// TwinCAT 3 PLC project TPR
// libraries:
//   Tc2_Standard, * (Beckhoff Automation GmbH)
//   Tc2_System, * (Beckhoff Automation GmbH)
//   Tc2_Utilities, * (Beckhoff Automation GmbH)
//   Tc3_Database, * (Beckhoff Automation GmbH)
//   Tc3_EventLogger, * (Beckhoff Automation GmbH)
//   Tc3_IotBase, * (Beckhoff Automation GmbH)
//   Tc3_Module, * (Beckhoff Automation GmbH)
// project tree:
//   Data types/ PrgData.TcDUT, frameData.TcDUT, ST_DataFromVision.TcDUT, ST_DataToVision.TcDUT, ST_ToolControl.TcDUT, ST_ToolData.TcDUT, ST_AdsTest.TcDUT
//   Global Variables/ CartControls.TcGVL, ErrorVar.TcGVL, Global_Variables.TcGVL
//   / PLC.TcTTO
//   POUs/ BackToZero.TcPOU, DB_Conn.TcPOU, ErrorHandle.TcPOU, GetCoordinates.TcPOU, LogProgram.TcPOU, MAIN.TcPOU, OnOffRobotCut.TcPOU, PcCom.TcPOU, P_Mqtt.TcPOU, RobotService.TcPOU, SendCoordinates.TcPOU, Tools.TcPOU
//   POUs/CONTROLs/ BlockTest.TcPOU, CalibCam1.TcPOU, CalibCam2.TcPOU, Control.TcPOU, ControlAuto.TcPOU, ControlGrabAuto.TcPOU, ControlMoveToCalibPos.TcPOU
//   POUs/EasySql/F_FB/ FB_EasySql.TcPOU, F_Replace.TcPOU
//   POUs/FUNCTIONs/ CamControl_1.TcPOU, CamControl_2.TcPOU, PlaceCoordinates.TcPOU, RobotControl_1.TcPOU, ValveControl_1.TcPOU
//   POUs/SEQUENCEs/ DeleafPlace.TcPOU, FindJoint.TcPOU, GetStem.TcPOU, GrabJoint.TcPOU, GrabStem.TcPOU, MoveOnStem.TcPOU
//   POUs/SQL/00_TestData/ P_SqlGeneratTestData.TcPOU
//   POUs/SQL/01_Insert/ P_SqlInsert.TcPOU, P_SqlInsertLog.TcPOU, P_SqlInsertRowConstructor.TcPOU, P_SqlInsertUnionAll.TcPOU, P_SqlInsertAlarmLog.TcPOU
//   POUs/SQL/02_Delete/ P_SqlDelete.TcPOU
//   POUs/SQL/03_Select/ P_SqlSelect.TcPOU, P_SqlSelectAlarmLog.TcPOU, P_SqlSelectCurrent.TcPOU, P_SqlSelectAlarm.TcPOU, P_SqlSelectTop.TcPOU, P_SqlSelectRecipe.TcPOU, P_SqlSelectFrame.TcPOU, ST_SelectAlarmStruct.TcDUT, ST_SelectAlarmLogStruct.TcDUT, ST_SelectFrameStruct.TcDUT, ST_SelectCurrentStruct.TcDUT, ST_SelectStruct.TcDUT, ST_SelectRecipeStruct.TcDUT
//   POUs/SQL/04_Update/ P_SqlUpdate.TcPOU, P_SqlUpdateAlarmLog.TcPOU
//   POUs/SQL/05_Count/ P_SqlCount.TcPOU
//   POUs/SQL/06_Sum/ P_SqlSum.TcPOU
// real-time tasks:
//   TASK PLC: cycle T#10ms, priority 1, ADS port 350
// I/O:
//   DEVICE Device 1 (Beckhoff CCAT)
//   DEVICE Device 2 (EtherCAT), AmsNetId 192.168.56.1.3.1
//     Term 1 (EK1200) [EK1200-5000 EtherCAT Power supply (2A E-Bus)]
//       Term 2 (EL1859) [EL1859 8Ch. Dig. Input 24V, 3ms, 8Ch. Dig. Output 24V, 0.5A]
//       Term 3 (EL2809) [EL2809 16Ch. Dig. Output 24V, 0.5A]
//       Term 4 (EL5151) [EL5151 1Ch. Inc. Encoder]
//       Term 5 (EL6751) [EL6751 CANopen Master]
//       Term 6 (EL9011) [EL9011 End Terminal]
//   DEVICE Device 3 (EL6751), AmsNetId 192.168.56.1.4.1
//     Box 7 (CX2xxx CANopen Slave)
// variable links:
//   TPR/TPR Instance <-> Device 2 (EtherCAT)/Term 1 (EK1200)/Term 2 (EL1859)
//     PLC Inputs/Global_Variables.bGripSensorStop <-> Channel 2/Input
//     PLC Inputs/OnOffRobotCut.bStartBotton <-> Channel 1/Input
//     PLC Outputs/Tools.qValve1 <-> Channel 9/Output
//     PLC Outputs/Tools.qValve2 <-> Channel 10/Output
//     PLC Outputs/Tools.qValve3 <-> Channel 11/Output
//     PLC Outputs/Tools.qValve4 <-> Channel 13/Output
//     PLC Outputs/Tools.qValve5 <-> Channel 12/Output
//   TPR/TPR Instance <-> Device 2 (EtherCAT)/Term 1 (EK1200)/Term 3 (EL2809)
//     PLC Outputs/CartControls.CartBackward <-> Channel 8/Output
//     PLC Outputs/CartControls.CartDown <-> Channel 6/Output
//     PLC Outputs/CartControls.CartForward <-> Channel 7/Output
//     PLC Outputs/CartControls.CartUp <-> Channel 5/Output
//     PLC Outputs/CartControls.WheelsChange <-> Channel 10/Output
//     PLC Outputs/Tools.qMotorDirection <-> Channel 2/Output
//     PLC Outputs/Tools.qMotorRun <-> Channel 1/Output
//   TPR/TPR Instance <-> Device 2 (EtherCAT)/Term 1 (EK1200)/Term 4 (EL5151)
//     PLC Inputs/Global_Variables.uiSignalInEncoderCount <-> ENC Inputs/Counter value
//     PLC Outputs/Global_Variables.bSetCounter <-> ENC Outputs/Control/Set counter
//     PLC Outputs/Global_Variables.uiSetCounterValue <-> ENC Outputs/Set counter value
//   TPR/TPR Instance <-> Device 3 (EL6751)/Box 7 (CX2xxx CANopen Slave)
//     PLC Inputs/ErrorVar.ErrorNum <-> TxPDO 4/Inputs/Byte_Input_30
//     PLC Inputs/ErrorVar.ErrorNum @bit 8 <-> TxPDO 4/Inputs/Byte_Input_31
//     PLC Inputs/ErrorVar.ErrorNum @bit 16 <-> TxPDO 4/Inputs/Byte_Input_32
//     PLC Inputs/ErrorVar.WhichRobot <-> TxPDO 4/Inputs/Byte_Input_29
//     PLC Inputs/Global_Variables.uiSignalIn2 <-> TxPDO 1/Inputs/Byte_Input_2
//     PLC Inputs/Global_Variables.uiSignalIn4 <-> TxPDO 1/Inputs/Byte_Input_4
//     PLC Inputs/Global_Variables.uiSignalInA <-> TxPDO 2/Inputs/Byte_Input_13
//     PLC Inputs/Global_Variables.uiSignalInA @bit 8 <-> TxPDO 2/Inputs/Byte_Input_14
//     PLC Inputs/Global_Variables.uiSignalInAck <-> TxPDO 1/Inputs/Byte_Input_5
//     PLC Inputs/Global_Variables.uiSignalInE <-> TxPDO 2/Inputs/Byte_Input_15
//     PLC Inputs/Global_Variables.uiSignalInE @bit 8 <-> TxPDO 2/Inputs/Byte_Input_16
//     PLC Inputs/Global_Variables.uiSignalInOrientation <-> TxPDO 3/Inputs/Byte_Input_19
//     PLC Inputs/Global_Variables.uiSignalInR <-> TxPDO 3/Inputs/Byte_Input_17
//     PLC Inputs/Global_Variables.uiSignalInR @bit 8 <-> TxPDO 3/Inputs/Byte_Input_18
//     PLC Inputs/Global_Variables.uiSignalInRobotFail <-> TxPDO 4/Inputs/Byte_Input_27
//     PLC Inputs/Global_Variables.uiSignalInShared <-> TxPDO 2/Inputs/Byte_Input_12
//     PLC Inputs/Global_Variables.uiSignalInToolAck <-> TxPDO 3/Inputs/Byte_Input_20
//     PLC Inputs/Global_Variables.uiSignalInX <-> TxPDO 3/Inputs/Byte_Input_21
//     PLC Inputs/Global_Variables.uiSignalInX @bit 8 <-> TxPDO 3/Inputs/Byte_Input_22
//     PLC Inputs/Global_Variables.uiSignalInY <-> TxPDO 3/Inputs/Byte_Input_23
//     PLC Inputs/Global_Variables.uiSignalInY @bit 8 <-> TxPDO 3/Inputs/Byte_Input_24
//     PLC Inputs/Global_Variables.uiSignalInZ <-> TxPDO 4/Inputs/Byte_Input_25
//     PLC Inputs/Global_Variables.uiSignalInZ @bit 8 <-> TxPDO 4/Inputs/Byte_Input_26
//     PLC Inputs/OnOffRobotCut.uiSignalIn1 <-> TxPDO 1/Inputs/Byte_Input_1
//     PLC Inputs/OnOffRobotCut.uiSignalIn3 <-> TxPDO 1/Inputs/Byte_Input_3
//     PLC Outputs/ErrorVar.CancelAlarm <-> RxPDO 4/Outputs/Byte_Output_32
//     PLC Outputs/ErrorVar.gSeverity <-> RxPDO 4/Outputs/Byte_Output_31
//     PLC Outputs/Global_Variables.gJointFound <-> RxPDO 3/Outputs/Byte_Output_18
//     PLC Outputs/Global_Variables.gTomatoHeading <-> RxPDO 4/Outputs/Byte_Output_29
//     PLC Outputs/Global_Variables.iImageZone <-> RxPDO 2/Outputs/Byte_Output_16
//     PLC Outputs/Global_Variables.uiCalibImgCount <-> RxPDO 2/Outputs/Byte_Output_14
//     PLC Outputs/Global_Variables.uiSignalOut1 <-> RxPDO 1/Outputs/Byte_Output_1
//     PLC Outputs/Global_Variables.uiSignalOut2 <-> RxPDO 1/Outputs/Byte_Output_2
//     PLC Outputs/Global_Variables.uiSignalOut3 <-> RxPDO 1/Outputs/Byte_Output_3
//     PLC Outputs/Global_Variables.uiSignalOutA <-> RxPDO 2/Outputs/Byte_Output_9
//     PLC Outputs/Global_Variables.uiSignalOutBoxHeight <-> RxPDO 4/Outputs/Byte_Output_28
//     PLC Outputs/Global_Variables.uiSignalOutBoxLength <-> RxPDO 4/Outputs/Byte_Output_26
//     PLC Outputs/Global_Variables.uiSignalOutBoxWidth <-> RxPDO 4/Outputs/Byte_Output_27
//     PLC Outputs/Global_Variables.uiSignalOutControl <-> RxPDO 1/Outputs/Byte_Output_8
//     PLC Outputs/Global_Variables.uiSignalOutE <-> RxPDO 2/Outputs/Byte_Output_10
//     PLC Outputs/Global_Variables.uiSignalOutOrientation <-> RxPDO 2/Outputs/Byte_Output_12
//     PLC Outputs/Global_Variables.uiSignalOutPackingMode <-> RxPDO 4/Outputs/Byte_Output_25
//     PLC Outputs/Global_Variables.uiSignalOutPick <-> RxPDO 3/Outputs/Byte_Output_17
//     PLC Outputs/Global_Variables.uiSignalOutR <-> RxPDO 2/Outputs/Byte_Output_11
//     PLC Outputs/Global_Variables.uiSignalOutShared <-> RxPDO 1/Outputs/Byte_Output_7
//     PLC Outputs/Global_Variables.uiSignalOutSpeedControl <-> RxPDO 2/Outputs/Byte_Output_13
//     PLC Outputs/Global_Variables.uiSignalOutTool <-> RxPDO 2/Outputs/Byte_Output_15
//     PLC Outputs/Global_Variables.uiSignalOutX <-> RxPDO 1/Outputs/Byte_Output_4
//     PLC Outputs/Global_Variables.uiSignalOutX2 <-> RxPDO 3/Outputs/Byte_Output_19
//     PLC Outputs/Global_Variables.uiSignalOutX2 @bit 8 <-> RxPDO 3/Outputs/Byte_Output_20
//     PLC Outputs/Global_Variables.uiSignalOutY <-> RxPDO 1/Outputs/Byte_Output_5
//     PLC Outputs/Global_Variables.uiSignalOutY2 <-> RxPDO 3/Outputs/Byte_Output_21
//     PLC Outputs/Global_Variables.uiSignalOutY2 @bit 8 <-> RxPDO 3/Outputs/Byte_Output_22
//     PLC Outputs/Global_Variables.uiSignalOutZ <-> RxPDO 1/Outputs/Byte_Output_6
//     PLC Outputs/Global_Variables.uiSignalOutZ2 <-> RxPDO 3/Outputs/Byte_Output_23
//     PLC Outputs/Global_Variables.uiSignalOutZ2 @bit 8 <-> RxPDO 3/Outputs/Byte_Output_24

CONFIGURATION TPR
    RESOURCE PLC ON TwinCAT3
        TASK PLC(INTERVAL := T#10ms, PRIORITY := 1);
        PROGRAM MAIN WITH PLC : MAIN;
    END_RESOURCE
END_CONFIGURATION

// ---- Data types/PrgData.TcDUT
TYPE PrgData :
STRUCT
	usiRecipe 			: USINT;
	usiNewRecipe		: USINT := 1;
	usiNewVelocity		: USINT;
	usiProgram			: USINT;
	usiNewProgram		: USINT;
	
	uiValveDelay		: UINT;
	uiCartheight		: UINT;
	usiVelocity			: USINT;
	usiOpMode			: USINT;
	usiPackingPattern	: USINT;
	usiImageRetryNo		: USINT;	
	

END_STRUCT
END_TYPE

// ---- Data types/frameData.TcDUT
TYPE frameData :
STRUCT
	ct_x	: DINT := 0;
	ct_y	: DINT := 0;
	ct_z	: DINT := 0;
	ct_a	: DINT := 0;
	ct_e	: DINT := 0;
	ct_r	: DINT := 0;
	
	cw_x	: DINT := 0;
	cw_y	: DINT := 0;
	cw_z	: DINT := 0;
	cw_a	: DINT := 0;
	cw_e	: DINT := 0;
	cw_r	: DINT := 0;
	
	pt_x	: DINT := 0;
	pt_y	: DINT := 0;
	pt_z	: DINT := 0;
	pt_a	: DINT := 0;
	pt_e	: DINT := 0;
	pt_r	: DINT := 0;
	
	pw_x	: DINT := 0;
	pw_y	: DINT := 0;
	pw_z	: DINT := 0;
	pw_a	: DINT := 0;
	pw_e	: DINT := 0;
	pw_r	: DINT := 0;

END_STRUCT
END_TYPE

// ---- Data types/ST_DataFromVision.TcDUT
TYPE ST_DataFromVision :
STRUCT

	CmdIdIn 			: DWORD;   		(*ECHO if Current ID Byte 1,2,3,4*)

								(*CMD 2-7:					CMD 8-9:							CMD 10:					CMD 11:			*)
	ResultPar1 		: INT;               	(*1: Done,    255: Failed		0: Searching,   1: Stop 255: Error            	P X						Crus X				*)	(* ResultPar1 Byte  7 	&	8 	*)
	ResultPar2 		: INT;		(*														P Y						Crus Y				*)	(* ResultPar2 Byte  9	&   	10 	*)
	ResultPar3 		: INT;		(*														P Z						Crus Z				*)	(* ResultPar3 Byte  11 	& 	12 	*)
	ResultPar4 		: INT;		(*														P Z0 rotation				Stem heading angle	*)	(* ResultPar4 Byte  13 	& 	14 	*)
	ResultPar5 		: INT;		(*														P Y   rotation									*)	(* ResultPar5 Byte  15 	& 	16 	*)
	ResultPar6 		: INT;		(*														P Z1 rotation									*)	(* ResultPar6 Byte  17 	& 	18 	*)
	ResultPar7 		: INT;		(*														P2 rotation around Z							*)	(* ResultPar7 Byte  19 	& 	20 	*)
	(* ResultPar9 Byte  23 	& 	24 	*)

	(*				Cam 1 information																Cam 2 information
		ResultPar1:	Stem pos Low 	X															Pos 		X
		ResultPar2:	Stem pos Low 	Y															Pos 		Y
		ResultPar3:	Stem pos Low 	Z															Pos 		Z
		ResultPar4:	Lowest tomato  	X															Rotation Z0			(Stem heading angle)
		ResultPar5:	Lowest tomato  	Y															Rotation Y			(Stem heading angle)
		ResultPar6:	Lowest tomato  	Z															Rotation Z1			(Stem heading angle)
		ResultPar7:	Rotation around Z	-	Angle between vector from stem to lowest tomato and X-axis		P2 rotation around Z						
	*)

	gStemFound	 	: BYTE; 	(*0: Not found 1: Found 255: timeout  Byte 5*)	(* Byte 5 *)
	gJointFound		: BYTE;		(*0: Not found 1: Found 255: timeout  Byte 6 *)	(* Byte 6 *)
	gTrussFound		: BYTE; 	(*0: Not found 1: Found 255: timeout  Byte 6 *)	(* Byte 7 *)
	gTomatoFound	: BYTE;		(*0: Not found 1: Found 255: timeout  Byte 6 *)	(* Byte 8 *)

	CmdInProcess	: BYTE;     	(*ECHO of current CMD Byte 0*)
END_STRUCT
END_TYPE

// ---- Data types/ST_DataToVision.TcDUT
TYPE ST_DataToVision :
STRUCT
	CmdIdOut	: DWORD;	(*
									0	Nothing
									1	Hello World
									2	Calib Cam 1 Start
									3	New Pos Calib Cam 1
									4	End Calib Cam 1
									5	Calib Cam 2 Start
									6	New Pos Calib Cam 2
									7	End Calib Cam 2
									8	Start  Stop At Plant Check (Cam 1)
									9	Stop Check (Cam 1)
									10	Request Plant Data (Cam 1)
									11	Manual Plant Data (Cam 1)
									12	Request Plant Data (Cam 2)
									13	Manual Plant Data (Cam 2)
									14	Restart
									15	Shutdown
									20	Distance check
								Byte 1,2,3,4
								*)


	CoordXR1G 	: INT; (*Update continously, R1: Cutter robot, G: global vehicle frame, Byte 6,7*)
	CoordYR1G  	: INT; (*Update continously, R1: Cutter robot, G: global vehicle frame, Byte 8,9*)
	CoordZR1G  	: INT; (*Update continously, R1: Cutter robot, G: global vehicle frame, Byte 10,11*)

	CoordXR2G  	: INT; (*Update continously, R2: Cutter robot, G: global vehicle frame, Byte 12,13*)
	CoordYR2G  	: INT; (*Update continously, R2: Cutter robot, G: global vehicle frame, Byte 14,15*)
	CoordZR2G  	: INT; (*Update continously, R2: Cutter robot, G: global vehicle frame, Byte 16,17*)

	CoordRRA  	: INT; (*Update continously, R2: Cutter robot, T: R2 TCP frame, Byte 18,19*)
	CoordRRE 	: INT; (*Update continously, R2: Cutter robot, T: R2 TCP frame, Byte 20,21*)
	CoordRRR 	: INT; (*Update continously, R2: Cutter robot, T: R2 TCP frame, Byte 22,23*)
	CmdByte 	: BYTE; (*Commands to Pc Byte 0*)
	ResultRead 	: BYTE; (*0: waiting 1: read Byte 5*)		(* Bruges ikke *)
END_STRUCT
END_TYPE

// ---- Data types/ST_ToolControl.TcDUT
TYPE ST_ToolControl :
STRUCT



END_STRUCT
END_TYPE

// ---- Data types/ST_ToolData.TcDUT
TYPE ST_ToolData :
STRUCT
END_STRUCT
END_TYPE

// ---- Data types/ST_AdsTest.TcDUT
TYPE ST_AdsTest :
STRUCT
	byteValue	:	BYTE := 255;
	wordValue	:	WORD := 2300;
	dwordValue	:	DWORD := 10;
	sintValue	:	SINT := -50;
	intValue	:	INT := 16555;
	dintValue	:	DINT := 65345;
	realValue 	:	REAL := 150.345;
	lrealValue	:	LREAL := -50.50;	

END_STRUCT
END_TYPE

// ---- POUs/SQL/03_Select/ST_SelectAlarmStruct.TcDUT
TYPE ST_SelectAlarmStruct :
STRUCT
	alarmId				: DINT;
	alarmDesc			: STRING(200);
	alarmCause			: STRING(500);
	alarmRemedy			: STRING(500);
END_STRUCT
END_TYPE

// ---- POUs/SQL/03_Select/ST_SelectAlarmLogStruct.TcDUT
TYPE ST_SelectAlarmLogStruct :
STRUCT
	dtTime				: DT;
	alarmId				: DINT;
	deviceWhich			: STRING(50);
END_STRUCT
END_TYPE

// ---- POUs/SQL/03_Select/ST_SelectFrameStruct.TcDUT
TYPE ST_SelectFrameStruct :
STRUCT
	sId	: STRING(45);
	diX	: DINT;
	diY	: DINT;
	diZ	: DINT;
	diA	: DINT;
	diE	: DINT;
	diR	: DINT;
END_STRUCT
END_TYPE

// ---- POUs/SQL/03_Select/ST_SelectCurrentStruct.TcDUT
TYPE ST_SelectCurrentStruct :
STRUCT
	recipe_id				: DINT;
	program_no				: DINT;
END_STRUCT
END_TYPE

// ---- POUs/SQL/03_Select/ST_SelectStruct.TcDUT
TYPE ST_SelectStruct :
STRUCT
	id: DINT;
	username: STRING(199);
	password: STRING(199);
END_STRUCT
END_TYPE

// ---- POUs/SQL/03_Select/ST_SelectRecipeStruct.TcDUT
TYPE ST_SelectRecipeStruct :
STRUCT
	recipe_id				: DINT;
	recipe_name				: STRING(199);
	recipe_velocity			: DINT;
	Operation_mode_id		: DINT;
	packing_pattern_id		: DINT;
	recipe_valve_delay		: DINT;
	recipe_cart_height		: DINT;
	recipe_image_retry_no	: DINT;
END_STRUCT
END_TYPE

// ---- Global Variables/CartControls.TcGVL
{attribute 'qualified_only'}
VAR_GLOBAL
	CartUp 			AT %Q*: BOOL := FALSE;		(* Lift kører op *)
	CartDown 		AT %Q*: BOOL := FALSE;		(* Lift kører ned *)
	CartForward 	AT %Q*: BOOL := FALSE;		(* Vogn kører fremad *)
	CartBackward 	AT %Q*: BOOL := FALSE;		(* Vogn kører bagud*)
	WheelsChange 	AT %Q*: BOOL := FALSE;		(* Hjul til sidelæns kørsel kører op/ned*)
END_VAR

// ---- Global Variables/ErrorVar.TcGVL
//{attribute 'qualified_only'}
VAR_GLOBAL
	ErrorNum 			AT %I*: DWORD; (* Error/warning received from the robots *)
	WhichRobot			AT %I*: BYTE; (* 1:Cut 2:Pick *)
	CancelAlarm			AT %Q*: BYTE; (* 0:Waiting for cancel alarm 1:Cancel Alarm*)
	gSeverity			AT %Q*: BYTE; (* 0:No Alarm 1:Warning 2:Error *)
END_VAR

// ---- Global Variables/Global_Variables.TcGVL
//{attribute 'Tc2GvlVarNames'}
 VAR_GLOBAL
	bReady: BOOL := FALSE;
	(* ------------------Binary values to commands--------------- *)
	Send_pos:					BYTE := 1;
	Send_pos_pick:				BYTE := 2;
	Move_to_idle:				BYTE := 3;
	Slave_to_image_pos:			BYTE := 4;
	Slave_to_grab_pos:			BYTE := 5;
	Slave_to_place_pos:			BYTE := 6;
	Master_move_to_stem:		BYTE := 7;
	Master_move_on_stem:		BYTE := 8;
	Master_move_from_stem:		BYTE := 9;
	Slave_move_from_pick:		BYTE := 10;
	Set_Velocity:				BYTE := 11;
	getCurrentCutCoords:		BYTE := 12;
	getCurrentPickCoords:		BYTE := 13;
	CalibCamOne:				BYTE := 14;
	CalibCamTwo:				BYTE := 15;
	Master_rotate_on_stem: 		BYTE := 16;
	Pick_Move_To_Pos: 			BYTE := 17;
	MOVE_CUT_TO_POS:			BYTE := 18;
	Pick_Move_From_Place:		BYTE := 19;
	Pick_Place_Cut_Move:		BYTE := 20;
	Pick_Trunk_Image:			BYTE := 21;
	DELEAF_IMAGE_PROGRAM:		BYTE := 22;
	INSERT_TO_PATH:				BYTE := 23;
	MOVE_ON_STEM_IMAGE:			BYTE := 24;
	PLACE_DELEAF:				BYTE := 25;
	Send_two_pos:				BYTE := 26;
	IMAGE_POS_GRAB_STEM:		BYTE := 27;
	RETRY_GRAB_STEM:			BYTE := 28;
	ROBOT_SERVICE:				BYTE := 29;
	CUT_BACK_TO_ZERO:			BYTE := 30;
	PICK_BACK_TO_ZERO:			BYTE := 31;
	CUT_TO_IDLE:				BYTE := 32;
	PICK_TO_IDLE:				BYTE := 33;

	FB_SEND_POS: 				RobotControl_1;
	FB_MOVE_TO_IDLE:			RobotControl_1;
	FB_IMAGE_POS: 				RobotControl_1;
	FB_PICK_GRAB:				RobotControl_1;
	FB_PICK_PLACE:				RobotControl_1;
	FB_PICK_MOVE_FROM_PICK:		RobotControl_1;
	FB_CUT_TO_STEM:				RobotControl_1;
	FB_CUT_ON_STEM:				RobotControl_1;
	FB_CUT_FROM_STEM:			RobotControl_1;
	FB_SET_VELOCITY:			RobotControl_1;
	FB_GET_CUT_COORD:			RobotControl_1;
	FB_GET_PICK_COORD:			RobotControl_1;
	FB_CALIB_CAM_ONE:			RobotControl_1;
	FB_CALIB_CAM_TWO:			RobotControl_1;
	FB_PICK_FROM_PLACE:			RobotControl_1;
	FB_PICK_TRUNK_IMAGE:		RobotControl_1;
	FB_PICK_DELEAF_PROGRAM:		RobotControl_1;
	FB_COMOVE_IMAGE:			RobotControl_1;
	FB_PLACE_DELEAF:			RobotControl_1;
	FB_SEND_TWO_POS:			RobotControl_1;
	FB_IMAGE_GRAB:				RobotControl_1;
	FB_RETRY_GRAB_STEM:			RobotControl_1;
	FB_CUT_TO_ZERO:				RobotControl_1;
	FB_PICK_TO_ZERO:			RobotControl_1;
	FB_ROBOT_SERVICE:			RobotControl_1;
	FB_CUT_TO_IDLE:				RobotControl_1;
	FB_PICK_TO_IDLE:				RobotControl_1;

	(* -------------------------Modbus to HMI------------------------- *)
	(* Control *)
	bStart 				AT %MX50.0: 	BOOL; 				(*%MW12313:X0*)
	bStartBottonHMI		AT %MX50.4: 	BOOL;				(*%MW12313:X4*)
	bStop 				AT %MX50.1: 	BOOL; 				(*%MW12313:X1*)
	bAlarmState 		AT %MX50.2: 	BOOL; 				(*%MW12313:X2*)
	uiStatus 			AT %MB10: 		UINT; 				(*%MW12293*)

	(* Status *)
	bRobotPickStatus	AT %MX50.5:		BOOL := FALSE;		(*%MW12313:X5*)
	bRobotCutStatus		AT %MX50.6:		BOOL := FALSE;		(*%MW12313:X6*)
	bPLCStatus			AT %MX50.7: 	BOOL := FALSE;		(*%MW12313:X7*)
	NewbPLCStatus 		: 	BOOL;
	NewbRobotCutStatus	:	BOOL;
	NewbRobotPickStatus	:	BOOL;

	(* Alarm *)
	bAckAlarm 			AT %MX50.3: 	BOOL; 				(*%MW12313:X3*)
	uiAlarm 			AT %MB12: 		UDINT := 0;			(*%MW12294*)
	bRobotAlarm			AT %MX56.0:		BOOL;				(*%MW12314:X0*)

	(* Speed *)
	uiSpeedSetting 		AT %MB24: 		USINT := 1; 			(*%MW12300*)

	(* Program *)
	uiprogNo 			AT %MB20: 		USINT := 0; 			(*%MW12298 *)   (* 0:No Program	1:CalibCam1		2:CalibCam2		3:Move to calib pos	4:Auto (NO adaptive )	5:GRAB AUTO*)
	sprogName 			AT %MB100: 		STRING := 'No Program'; 		(*%MB12338*)
	sprogNameArray:  	ARRAY[1..15] OF STRING :=[ 'No Program', 'Calib Cam 1', 'Calib Cam 2', 'Move to calib pos',  'Auto', 'GRAB AUTO'];

	uimodeNo			AT %MB22:		USINT := 0;			(* %MW12299 *)  (* 0: Both			1:Tomato cutting	2:Deleafing *)
	smodeName 			AT %MB150:		STRING := 'Both';		(* %MW12363 *)
	smodeNameArray: 	ARRAY[1..3] OF STRING :=[ 'Both', 'Tomato Cutting', 'Deleafing'];

	uiPackingModeNo 	AT %MB26:	USINT := 0;			(*%MW12301*)
	sPackingModeName 	AT %MB250: STRING :='DEFAULT';	(* %MW12413 *)
	sPackingModeNameArray: ARRAY[1..2] OF STRING :=[ 'DEFAULT', 'OTHER'];
	uiPackModeNo 		AT %Q*:BYTE;

	uiBoxLength			AT %MB28:	 UINT := 450;			(*%MW12302*)
	uiBoxWidth			AT %MB32:	UINT := 400;			(*%MW12304*)
	uiBoxHeight			AT %MB36:	UINT := 200;			(*%MW12306*)

	MasterState 		AT %MB200:	 INT := 0;				(*Master state*)

	(* PC control *)
	bHelloWorld				AT %MX52.0:	BOOL;		(*%MW12314:X0*)
	bCalibCamOneStart		AT %MX52.1:	BOOL;		(*%MW12314:X1*)
	bNewPosCalibCamOne	AT %MX52.2:	BOOL;		(*%MW12314:X2*)
	bEndCalibCamOne		AT %MX52.3:	BOOL;		(*%MW12314:X3*)
	bCalibCamTwoStart		AT %MX52.4:	BOOL;		(*%MW12314:X4*)
	bNewPosCalibCamTwo	AT %MX52.5:	BOOL;		(*%MW12314:X5*)
	bEndCalibCamTwo		AT %MX52.6:	BOOL;		(*%MW12314:X6*)
	bStartStopPlantCheck		AT %MX52.7:	BOOL;		(*%MW12314:X7*)
	bStopCheck				AT %MX54.0: BOOL;		(*%MW12315:X0*)
	bGetPlantDataCamOne	AT %MX54.1: BOOL;		(*%MW12315:X1*)
	bGetPlantDataCamTwo	AT %MX54.2: BOOL;		(*%MW12315:X2*)
	bRestart					AT %MX54.3: BOOL;		(*%MW12315:X3*)
	bShutdown				AT %MX54.4: BOOL;		(*%MW12315:X4*)
	bTestCamPointCam2		AT %MX54.5: BOOL;		(*%MW12315:X5*)
	bTestCamPointCam1		AT %MX54.6: BOOL;		(*%MW12315:X6*)

	bRobotServiceStart			AT %MX54.7: BOOL;		(*%MW12315:X7*)
	bRobotServiceStop : BOOL;
	
	bBackToZero			AT %MX56.0:	BOOL;		(*%MW12316:X0*)



	(* --------------------------------------------------FUNCTION BLOCKs-------------------------------------------------- *)
	FB_CAM_ONE_CONTROL:	CamControl_1;
	FB_CAM_TWO_CONTROL:	CamControl_2;

	FB_PLACE: 			PlaceCoordinates;
	FB_GET_STEM:		GetStem;
	FB_GRAB_STEM:		GrabStem;
	FB_MOVE_ON_STEM:	MoveOnStem;
	FB_FIND_JOINT:		FindJoint;
	FB_GRAB_JOINT:		GrabJoint;
	FB_DELEAF_PLACE:	DeleafPlace;

	FB_OPEN_CUT : 		ValveControl_1;
	FB_CLOSE_CUT : 		ValveControl_1;
	FB_RELEASE_CUT :	ValveControl_1;
	FB_OPEN_PICK : 		ValveControl_1;
	FB_CLOSE_PICK : 	ValveControl_1;

	FB_LOAD_CUT: 		ValveControl_1;
	FB_DELOAD_CUT: 		ValveControl_1;

	FB_OPEN_GRIP: 		ValveControl_1;
	FB_CLOSE_GRIP: 		ValveControl_1;
	
	FB_BRAKE: 			ValveControl_1;

	(* --------------------------------------------------Shared variables-------------------------------------------------- *)

	(* REALS *)

	(* INTEGERS *)
	uiTrunkPos: 		UINT;				(* Stamme position	-->	Afstand i mm.															*)
	iBunchPosZ: 		UINT;
	iStemAngle:			INT;

	uiCutCoordX: 		UINT;
	uiCutCoordY: 		UINT;
	uiCutCoordZ: 		UINT;

	iStemPosX: 			UINT;				(* *)
	iStemPosY: 			UINT;				(* *)
	iStemPosZ: 			UINT;
	iRoll: 				INT;
	iPitch: 			UINT;
	iYaw:				INT;
	iPickAngle: 		INT;

	ImageRetryHeight:	INT;
	
	robotAlarmId:		UDINT;
	
	bAlarm:				BOOL;
	bAlarmAck:			BOOL;
	sDeviceWhich:		STRING;
	
	bLog:				BOOL;		// For logging of data
	tLogTime:			TON;		// Time for one sequence
	uiElapsedTime:		UINT;
	usiImageLog:		USINT;		// Counting number of images taken in a sequence
	usiStickoutCutLog:	USINT;		// For counting number of stick-outs
	usiRetryLog:		USINT;		// Number of retries in on control sequence
	usiImageRetry:		USINT;		// How many times to change image cnfg
	bLogSucces:			USINT;		// TRUE if success	-	FALSE if not
	
	


	(* --------------------------------------------------Tool parameters-------------------------------------------------- *)
	sToolControl	:STRING(45);


	(* Tool control AT %MX60	-	Modbus to HMI *)
	GbCloseCut				AT %MX60.0: BOOL;		(*%MW12318:X0*)
	GbOpenCut				AT %MX60.1: BOOL;		(*%MW12318:X1*)
	GbLoadCut				AT %MX60.2: BOOL;		(*%MW12318:X2*)
	GbClosePick				AT %MX60.3: BOOL;		(*%MW12318:X3*)
	GbOpenPick				AT %MX60.4: BOOL;		(*%MW12318:X4*)
	GbReleaseStem: BOOL;
	GbGripStem: BOOL;
	GbReleaseCut: BOOL;
	GbMotorIn: BOOL;
	GbHomeGripStem			AT %MX62.0: BOOL;		(*%MW12319:X0*)
	GbCloseGrip				AT %MX60.6: BOOL;		(*%MW12318:X6*)
	GbOpenGrip				AT %MX60.5: BOOL;		(*%MW12318:X5*)
	GbCancelAlarm: BOOL;
	bAck: BOOL;							(* Acknowledge Tool kommando *)
	bHomeDone: BOOL;
	GbDeloadCut				AT %MX60.7: BOOL;		(*%MW12318:X7*)

	Cam					AT %MX62.3: BOOL;		(*%MW12319:X3*)
	bResetButton				AT %MX62.4: BOOL;		(*%MW12319:X4*)
	bResetButton2			AT %MX62.5: BOOL;		(*%MW12319:X5*)


	(* --------------------------------------------------Ethercat to Vision-------------------------------------------------- *)
	(*OutPut*)

	stDataToVision: ST_DataToVision;
	
	stAdsTest : ST_AdsTest;

	(*InPut*)
	stDataFromVision : ST_DataFromVision;

	(* Sent to Robot Cut *)
	gStemFound AT %Q* 	: BYTE;
	gJointFound AT %Q* 	: BYTE;
	gTomatoHeading AT %Q* 	: BYTE;




	gSendCmdPc : BOOL;
	gCmdIdPc : BOOL;
	gErrorCode : INT;
	gResetPcCom: BOOL;
	bPosSentToPcCom: BOOL;

	(* --------------------------------------------------PLC parameters-------------------------------------------------- *)
	(*Sendcoord*)
	GsendCoord: BOOL;
	GcoordSent: BOOL;
	GviX : INT;
	GviY: INT;
	GviZ: INT;
	GviA: INT;
	GviE: INT;
	GviR: INT;
	GviX2: INT;
	GviY2: INT;
	GviZ2: INT;
	GviPick: INT;

	uiToolState: UINT;

	bCalibCheck 		: BOOL;
	sNewCalib 			: STRING(45);
	sCalib 				: STRING(45);
	usiVisionCmd		: USINT;
	calibContinue 		: BOOL;
	allZero 			: BOOL;

	(* --------------------------------------------------OnOffRobotCut parameters-------------------------------------------------- *)
	bRobotConnect		: BOOL;
	bRobotDisconnect	: BOOL;
	(*Out*)
	bNoHold 			: BOOL;
	bNoDriveOff			: BOOL;
	bDriveOn 			: BOOL;

	(*In*)
	bNoAlarm 			: BOOL;
	bDriveOnState 		: BOOL;
	bStartNoHold 		: BOOL;

	uiSignalOut1 AT %Q*	: BYTE;			(* OnOffRobotCut Controls *)
	uiSignalOut2 AT %Q*	: BYTE;


	uiSignalOut3 AT %Q*	: BYTE;			(* $DIN[1017..1025]		01 = Calib cam 2 pos (1018)		02 = (1019)		03 = (1020) 		1023 ()*)

	(* --------------------------------------------------SendCoordinates parameters-------------------------------------------------- *)
	(*Inputs - Sendcoords*)
	uiSignalIn4 AT %I*: BYTE;			(* $FMI[4] på Robot Cut *)

	(*Outputs - Sendcoords*)
	uiSignalOutX AT %Q*: BYTE;
	uiSignalOutY AT %Q*: BYTE;
	uiSignalOutZ AT %Q*: BYTE;
	uiSignalOutShared AT %Q*: BYTE;
	uiSignalOutA AT%Q*: BYTE;
	uiSignalOutE AT %Q*: BYTE;
	uiSignalOutR AT %Q*: BYTE;
	uiSignalOutPick AT %Q*: BYTE;
	uiSignalOutOrientation AT %Q*: BYTE;
	uiSignalOutX2 AT %Q*:	INT;
	uiSignalOutY2 AT %Q*:	INT;
	uiSignalOutZ2 AT %Q*:	INT;
	uiSignalOutBoxWidth AT %Q*: BYTE;
	uiSignalOutBoxLength AT %Q*: BYTE;
	uiSignalOutBoxHeight AT %Q*: BYTE;
	uiSignalOutPackingMode AT %Q*: BYTE;

	iImageZone AT %Q*: BYTE;

	(* --------------------------------------------------GetCoordinates parameters-------------------------------------------------- *)
	(*Tcp Coord Input - Getcoord*)
	uiSignalInX AT %I*: INT;
	uiSignalInY AT %I*: INT;
	uiSignalInZ AT %I*: INT;
	uiSignalInShared AT %I*: BYTE;
	uiSignalInA AT%I*: INT;
	uiSignalInE AT %I*: INT;
	uiSignalInR AT %I*: INT;
	uiSignalInOrientation AT %I*: BYTE;
	getPickCoords: BOOL;
	getCutCoords: BOOL;

	GgetCoord: BOOL;
	currentRobotX: INT;
	currentRobotY: INT;
	currentRobotZ: INT;
	currentRobotA: INT;
	currentRobotE: INT;
	currentRobotR: INT;
	PickCoord: BOOL;
	CutCoord: BOOL;
	bGetCoordDone: BOOL := FALSE;

	(*Output - Calib*)
	uiCalibImgCount AT %Q*: BYTE;			(* $FMI[14] på Robot Cut *)

	(*Inputs*)
	uiSignalIn2 AT %I*: BYTE;				(* DOUT[1009..1016]:	1016: GRAB FAIL *)
	uiSignalInAck AT %I*: BYTE;			(* $FMO[5] på Robot Cut *)
	uiSignalInToolAck AT %I*: BYTE;		(* $DOUT[1041..1048] på Robot Cut *)

	(*Outputs*)
	uiSignalOutControl AT %Q*: BYTE;		(* $FMI[8]  på Robot Cut *)
	uiSignalOutSpeedControl AT %Q*: BYTE;
	uiSignalOutTool AT %Q*: BYTE;		(* $DIN[0..0] på Robot Cut 		00=	Load Cut		01 =	Release Cut		02 = Open Cut		03 = Close Cut		04 = Open Pick		05 = Close Pick		07 = *)

	startCalibCam1: BOOL;
	startCalibCam2: BOOL;


	iEncoderCount: INT := 0;
	uiSignalInEncoderCount AT %I*: UDINT;
	bGripSensorStop AT %I*: BOOL;
	bSetCounter AT %Q*: BOOL;
	uiSetCounterValue AT %Q*: UDINT := 10000;
	uiDistToGrab: INT;				(* Measure in mm. *)
	next5:  BOOL;
	WaitGrip: TON;

	adstest : DINT := 0;

	(* Sensors *)
	bCutSensor:		 		BOOL;
	bPickSensor:			BOOL;
	bJorisSensor:			BOOL;
	
	PROGRAM_DATA 	: PrgData;
	FRAME_DATA		: frameData;

	bGetCutCoordDone: BOOL;
	gStopped: BOOL;
	
	uiSignalInRobotFail AT %I*: BYTE;
	
END_VAR


VAR_GLOBAL PERSISTENT
	arrPrograms: ARRAY [0..99] OF PrgData;
	stAktPrg AT %MB1000: PrgData;

END_VAR

// ---- POUs/MAIN.TcPOU
PROGRAM MAIN
VAR		

	iAlive : 						INT;
	ControlState: 					INT;
	ControlMoveToCalibPosState: 	INT;
	CalibCam1State: 				INT;
	CalibCam2State: 				INT;
	ToolsState: 					INT;
	ControlGrabAutoState: 			INT;

	bStopped: 					BOOL;
	bStopFlag: BOOL;

	trig:							R_TRIG;

	ControlAutoState: INT;
	ControlInternalState: INT;
	bService: BOOL;
	BlockTestState: INT;
	FB_MOVE_ON_STEM_STATE: INT;
	FB_GRAB_STEM_STATE: INT;
	FB_GRAB_JOINT_STATE: INT;
	turnOn: BOOL;
END_VAR
VAR_INPUT
	FB_GET_STEM_STATE: INT;
	FB_FIND_JOINT_STATE: INT;
END_VAR
VAR_OUTPUT
	FB_DELEAF_STATE: INT;
END_VAR

iAlive := iAlive + 1;

///////////////////////////// INIT Function blocks to communication /////////////////////////////
P_Mqtt();		// For pub/sub information to/from mosquitto broker


P_SqlGeneratTestData();

P_SqlSelect();
P_SqlSelectRecipe();
P_SqlSelectCurrent();
P_SqlSelectAlarm();
P_SqlSelectAlarmLog();
P_SqlSelectFrame();
P_SqlSelectTop();
P_SqlInsert();
P_SqlInsertAlarmLog();
P_SqlInsertLog();
P_SqlInsertRowConstructor();
P_SqlUpdate();
P_SqlUpdateAlarmLog();
P_SqlInsertRowConstructor();
P_SqlInsertUnionAll();
P_SqlDelete();
P_SqlCount();
P_SqlSum();

DB_Conn();

///////////////////////////// INIT sequences /////////////////////////////

OnOffRobotCut();
IF  OnOffRobotCut.State <> OnOffRobotCut.NewState THEN
	OnOffRobotCut.State := OnOffRobotCut.NewState;
END_IF

LogProgram();
IF  LogProgram.State <> LogProgram.NewState THEN
	LogProgram.State := LogProgram.NewState;
END_IF

Control();
IF Control.InternalState <> Control.InternalNewState THEN
	 Control.InternalState :=  Control.InternalNewState;
END_IF
IF Control.State <> Control.NewState THEN
	Control.State := Control.NewState;
END_IF

ControlAuto();
IF ControlAuto.State <> ControlAuto.NewState THEN
	ControlAuto.State := ControlAuto.NewState;
END_IF

ControlGrabAuto();
IF ControlGrabAuto.State <> ControlGrabAuto.NewState THEN
	ControlGrabAuto.State := ControlGrabAuto.NewState;
END_IF

ControlMoveToCalibPos();
IF ControlMoveToCalibPos.State <> ControlMoveToCalibPos.NewState THEN
	ControlMoveToCalibPos.State := ControlMoveToCalibPos.NewState;
END_IF

Tools();
IF  Tools.State <> Tools.NewState THEN
	Tools.State := Tools.NewState;
END_IF

SendCoordinates();
IF SendCoordinates.State <> SendCoordinates.NewState THEN
	SendCoordinates.State := SendCoordinates.NewState;
END_IF

PcCom();
IF  PcCom.State <> PcCom.NewState THEN
	PcCom.State := PcCom.NewState;
END_IF

ErrorHandle();
IF  ErrorHandle.State <> ErrorHandle.NewState THEN
	ErrorHandle.State := ErrorHandle.NewState;
END_IF

GetCoordinates();
IF GetCoordinates.State <> GetCoordinates.NewState THEN
	GetCoordinates.State := GetCoordinates.NewState;
END_IF

CalibCam1();
IF CalibCam1.State <> CalibCam1.NewState THEN
	CalibCam1.State := CalibCam1.NewState;
END_IF

CalibCam2();
IF CalibCam2.State <> CalibCam2.NewState THEN
	CalibCam2.State := CalibCam2.NewState;
END_IF

BackToZero();
IF BackToZero.State <> BackToZero.NewState THEN
	BackToZero.State := BackToZero.NewState;
END_IF

RobotService();
IF RobotService.State <> RobotService.NewState THEN
	RobotService.State := RobotService.NewState;
END_IF

BlockTest();
IF BlockTest.State <> BlockTest.NewState THEN
	BlockTest.State := BlockTest.NewState;
END_IF

(*Lukker griber ved opstart, så den ikke hænger fast i planterne on indkøring*)
IF NOT turnOn THEN 
	FB_CLOSE_GRIP.Execute := TRUE;
	IF FB_CLOSE_GRIP.Done THEN
		FB_CLOSE_GRIP.Execute := FALSE;
		turnOn := TRUE;
	END_IF
END_IF

IF BlockTest.State = 0 AND CalibCam1.State = 0 AND CalibCam2.State = 0 AND Control.State = 0 AND ControlAuto.State = 0 AND ControlGrabAuto.State = 0 AND ControlMoveToCalibPos.State = 0 AND Tools.State = 0 THEN
	allZero := TRUE;
ELSE
	allZero := FALSE;
END_IF

///////////////////////////// Reset sequence /////////////////////////////
IF bResetButton THEN
	bResetButton := FALSE;
	Control.NewState := 1000;

	ControlAuto.NewState := 1000;
	ControlMoveToCalibPos.NewState := 1000;
	CalibCam1.NewState := 1000;
	CalibCam2.NewState := 1000;
	ControlGrabAuto.NewState := 1000;
	Tools.NewState := 1000;

	BlockTest.NewState := 1000;

	FB_GET_STEM.				Execute := FALSE;
	FB_GRAB_STEM.				Execute := FALSE;
	FB_MOVE_ON_STEM.			Execute := FALSE;
	FB_FIND_JOINT.				Execute := FALSE;
	FB_GRAB_JOINT.				Execute := FALSE;
	FB_DELEAF_PLACE.			Execute := FALSE;

	FB_GET_STEM.				NewState := 1000;
	FB_GRAB_STEM.				NewState := 1000;
	FB_MOVE_ON_STEM.			NewState := 1000;
	FB_FIND_JOINT.				NewState := 1000;
	FB_GRAB_JOINT.				NewState := 1000;
	FB_DELEAF_PLACE.			NewState := 1000;


	FB_SEND_POS.				Execute := FALSE;
	FB_MOVE_TO_IDLE.			Execute := FALSE;
	FB_IMAGE_POS.				Execute := FALSE;
	FB_PICK_GRAB.				Execute := FALSE;
	FB_PICK_PLACE.				Execute := FALSE;
	FB_PICK_MOVE_FROM_PICK.	Execute := FALSE;
	FB_CUT_TO_STEM.			Execute := FALSE;
	FB_CUT_ON_STEM.			Execute := FALSE;
	FB_CUT_FROM_STEM.		Execute := FALSE;
	FB_SET_VELOCITY.			Execute := FALSE;
	FB_GET_CUT_COORD.		Execute := FALSE;
	FB_GET_PICK_COORD.		Execute := FALSE;
	FB_CALIB_CAM_ONE.			Execute := FALSE;
	FB_CALIB_CAM_TWO.			Execute := FALSE;
	FB_PICK_FROM_PLACE.		Execute := FALSE;
	FB_PICK_TRUNK_IMAGE.		Execute := FALSE;
	FB_PICK_DELEAF_PROGRAM.	Execute := FALSE;
	FB_ROBOT_SERVICE.		Execute := FALSE;


	FB_COMOVE_IMAGE.			Execute := FALSE;
	FB_PLACE_DELEAF.			Execute := FALSE;
	FB_SEND_TWO_POS.			Execute := FALSE;
	FB_IMAGE_GRAB.			Execute := FALSE;

	FB_RETRY_GRAB_STEM.		Execute := FALSE;

	FB_CUT_TO_ZERO.			Execute := FALSE;
	FB_PICK_TO_ZERO.		Execute := FALSE;

	FB_CAM_ONE_CONTROL.	Execute 	:= FALSE;
	FB_CAM_ONE_CONTROL.	NewState 	:= 1000;
	FB_CAM_TWO_CONTROL.	Execute 	:= FALSE;
	FB_CAM_TWO_CONTROL.	NewState 	:= 1000;
	
	gResetPcCom						:= TRUE;
	
	bService := FALSE;
	gResetPcCom := TRUE;

END_IF

IF bResetButton2 THEN
	bResetButton2 := FALSE;
	Control.NewState := 1000;
	BlockTest.NewState := 1000;
	ControlAuto.NewState := 1000;
	ControlMoveToCalibPos.NewState := 1000;
	CalibCam1.NewState := 1000;
	CalibCam2.NewState := 1000;
	ControlGrabAuto.NewState := 1000;
	Tools.NewState := 3000;

	bService := FALSE;

	FB_GET_STEM.				Execute := FALSE;
	FB_GRAB_STEM.				Execute := FALSE;
	FB_MOVE_ON_STEM.			Execute := FALSE;
	FB_FIND_JOINT.				Execute := FALSE;
	FB_GET_STEM.				Execute := FALSE;
	FB_GRAB_JOINT.				Execute := FALSE;
	FB_DELEAF_PLACE.			Execute := FALSE;

	FB_GET_STEM.				NewState := 1000;
	FB_GRAB_STEM.				NewState := 1000;
	FB_MOVE_ON_STEM.			NewState := 1000;
	FB_FIND_JOINT.				NewState := 1000;
	FB_GRAB_JOINT.				NewState := 1000;
	FB_DELEAF_PLACE.			NewState := 1000;

	FB_SEND_POS.				Execute := FALSE;
	FB_MOVE_TO_IDLE.			Execute := FALSE;
	FB_IMAGE_POS.				Execute := FALSE;
	FB_PICK_GRAB.				Execute := FALSE;
	FB_PICK_PLACE.				Execute := FALSE;
	FB_PICK_MOVE_FROM_PICK.	Execute := FALSE;
	FB_CUT_TO_STEM.			Execute := FALSE;
	FB_CUT_ON_STEM.			Execute := FALSE;
	FB_CUT_FROM_STEM.		Execute := FALSE;
	FB_SET_VELOCITY.			Execute := FALSE;
	FB_GET_CUT_COORD.		Execute := FALSE;
	FB_GET_PICK_COORD.		Execute := FALSE;
	FB_CALIB_CAM_ONE.			Execute := FALSE;
	FB_CALIB_CAM_TWO.			Execute := FALSE;
	FB_PICK_FROM_PLACE.		Execute := FALSE;
	FB_PICK_TRUNK_IMAGE.		Execute := FALSE;
	FB_PICK_DELEAF_PROGRAM.	Execute := FALSE;

	FB_ROBOT_SERVICE.		Execute := FALSE;


	FB_COMOVE_IMAGE.			Execute := FALSE;
	FB_PLACE_DELEAF.			Execute := FALSE;
	FB_SEND_TWO_POS.			Execute := FALSE;
	FB_IMAGE_GRAB.			Execute := FALSE;

	FB_RETRY_GRAB_STEM.		Execute := FALSE;

	FB_CUT_TO_ZERO.			Execute := FALSE;
	FB_PICK_TO_ZERO.			Execute := FALSE;

	FB_CAM_ONE_CONTROL.	Execute := FALSE;
	FB_CAM_TWO_CONTROL.	Execute := FALSE;


	gResetPcCom := TRUE;

END_IF

///////////////////////////// Stop/Pause sequence /////////////////////////////
IF bStop OR bStopped THEN
	uiStatus := 2;
	IF NOT bStopped THEN
		FB_GET_STEM_STATE 		:= FB_GET_STEM.State;
		FB_GRAB_STEM_STATE 		:= FB_GRAB_STEM.State;
		FB_MOVE_ON_STEM_STATE	:= FB_MOVE_ON_STEM.State;
		FB_FIND_JOINT_STATE 		:= FB_FIND_JOINT.State;
		FB_GRAB_JOINT_STATE		:= FB_GRAB_JOINT.State;
		FB_DELEAF_STATE 			:= FB_DELEAF_PLACE.State;

		FB_GET_STEM.NewState := 2000;
		FB_GRAB_STEM.NewState := 2000;
		FB_MOVE_ON_STEM.NewState := 2000;
		FB_FIND_JOINT.NewState := 2000;
		FB_GRAB_JOINT.NewState := 2000;
		FB_DELEAF_PLACE.NewState := 2000;

		ControlState 					:= Control.State;
		BlockTestState				:= BlockTest.State;

		ControlAutoState				:= ControlAuto.State;
		ControlMoveToCalibPosState 	:= ControlMoveToCalibPos.State;
		CalibCam1State 				:= CalibCam1.State;
		CalibCam2State 				:= CalibCam2.State;
		ControlGrabAutoState 			:= ControlGrabAuto.State;
		ToolsState 					:= Tools.State;

		BlockTest.State 					:= 2000;
		Control.State 						:= 2000;
		ControlAuto.NewState 				:= 2000;
		ControlMoveToCalibPos.NewState 	:= 2000;
		CalibCam1.NewState 				:= 2000;
		CalibCam2.NewState 				:= 2000;
		ControlGrabAuto.NewState 			:= 2000;
		Tools.NewState 					:= 2000;
		bStopped := TRUE;
	END_IF

	IF bStart THEN
		uiStatus := 1;

		FB_GET_STEM.NewState := FB_GET_STEM_STATE;
		FB_GRAB_STEM.NewState := FB_GRAB_STEM_STATE;
		FB_MOVE_ON_STEM.NewState := FB_MOVE_ON_STEM_STATE;
		FB_FIND_JOINT.NewState := FB_FIND_JOINT_STATE;
		FB_GRAB_JOINT.NewState := FB_GRAB_JOINT_STATE;
		FB_DELEAF_PLACE.NewState := FB_DELEAF_STATE;

		BlockTest.NewState := BlockTestState;
		Control.NewState := ControlState;
		ControlAuto.NewState := ControlAutoState;
		ControlMoveToCalibPos.NewState := ControlMoveToCalibPosState;
		CalibCam1.NewState := CalibCam1State;
		CalibCam2.NewState := CalibCam2State;
		ControlGrabAuto.NewState := ControlGrabAutoState;
		Tools.NewState := ToolsState;
		bStopped := FALSE;
	END_IF
END_IF


uiprogNo := PROGRAM_DATA.usiProgram;
IF PROGRAM_DATA.usiVelocity = 0 THEN
	uiSignalOutSpeedControl := 1;
ELSE
	uiSignalOutSpeedControl := PROGRAM_DATA.usiVelocity;
END_IF


///////////////////////////// FUNCTIONBLOCK CALL /////////////////////////////
FB_SEND_POS				(ControlType := 1,		Command := Send_pos,					Ack := uiSignalInAck);
FB_MOVE_TO_IDLE			(ControlType := 1,		Command := Move_to_idle,				Ack := uiSignalInAck);
FB_IMAGE_POS			(ControlType := 1,		Command := Slave_to_image_pos,			Ack := uiSignalInAck);
FB_PICK_GRAB			(ControlType := 1,		Command := Slave_to_grab_pos,			Ack := uiSignalInAck);
FB_PICK_PLACE			(ControlType := 1,		Command := Slave_to_place_pos,			Ack := uiSignalInAck);
FB_PICK_MOVE_FROM_PICK	(ControlType := 1,		Command := Slave_move_from_pick,		Ack := uiSignalInAck);
FB_CUT_TO_STEM			(ControlType := 1,		Command := Master_move_to_stem,			Ack := uiSignalInAck);
FB_CUT_ON_STEM			(ControlType := 1,		Command := Master_move_on_stem,			Ack := uiSignalInAck);
FB_CUT_FROM_STEM		(ControlType := 1,		Command := Master_move_from_stem,		Ack := uiSignalInAck);
FB_SET_VELOCITY			(ControlType := 1,		Command := Set_Velocity,				Ack := uiSignalInAck);
FB_GET_CUT_COORD		(ControlType := 1,		Command := getCurrentCutCoords,			Ack := uiSignalInAck);
FB_GET_PICK_COORD		(ControlType := 2,		Command := getCurrentPickCoords,		Ack := uiSignalInAck,		CoordX := stDataToVision.CoordXR2G,		CoordY := stDataToVision.CoordYR2G,		CoordZ := stDataToVision.CoordZR2G	);
FB_CALIB_CAM_ONE		(ControlType := 1,		Command := CalibCamOne,					Ack := uiSignalInAck);
FB_CALIB_CAM_TWO		(ControlType := 1,		Command := CalibCamTwo,					Ack := uiSignalInAck);
FB_PICK_FROM_PLACE		(ControlType := 1,		Command := Pick_Move_From_Place,		Ack := uiSignalInAck);
FB_PICK_TRUNK_IMAGE		(ControlType := 1,		Command := Pick_Trunk_Image,			Ack := uiSignalInAck);
FB_PICK_DELEAF_PROGRAM	(ControlType := 1,		Command := DELEAF_IMAGE_PROGRAM,		Ack := uiSignalInAck);
FB_COMOVE_IMAGE			(ControlType := 1,		Command := MOVE_ON_STEM_IMAGE,			Ack := uiSignalInAck);
FB_PLACE_DELEAF			(ControlType := 1,		Command := PLACE_DELEAF,				Ack := uiSignalInAck);
FB_SEND_TWO_POS			(ControlType := 1,		Command := Send_two_pos,				Ack := uiSignalInAck);
FB_IMAGE_GRAB			(ControlType := 1,		Command := IMAGE_POS_GRAB_STEM,			Ack := uiSignalInAck);
FB_RETRY_GRAB_STEM		(ControlType := 1,		Command := RETRY_GRAB_STEM,				Ack := uiSignalInAck);
FB_ROBOT_SERVICE		(ControlType := 1,		Command := ROBOT_SERVICE,				ACK := uiSignalInAck, Execute := bRobotServiceStart OR FB_ROBOT_SERVICE.Execute);
FB_CUT_TO_ZERO			(ControlType := 1,		Command := CUT_BACK_TO_ZERO,			Ack := uiSignalInAck);
FB_PICK_TO_ZERO			(ControlType := 1,		Command := PICK_BACK_TO_ZERO,			Ack := uiSignalInAck);
FB_CUT_TO_IDLE			(ControlType := 1,		Command := CUT_TO_IDLE,					Ack := uiSignalInAck);
FB_PICK_TO_IDLE			(ControlType := 1,		Command := PICK_TO_IDLE,				Ack := uiSignalInAck);

FB_PLACE(Offset := 140,		Box_length := uiBoxLength, 		Box_width := uiBoxWidth,	Box_height := uiBoxHeight,		Stem_length := 200,	Mode := uiPackingModeNo);

FB_GET_STEM();
FB_GRAB_STEM();
FB_MOVE_ON_STEM();
FB_FIND_JOINT();
FB_GRAB_JOINT();
FB_DELEAF_PLACE();


uiSignalOutBoxWidth		:= INT_TO_BYTE(uiBoxWidth/10);
uiSignalOutBoxLength 	:= INT_TO_BYTE(uiBoxLength/10);
uiSignalOutBoxHeight 	:= INT_TO_BYTE(uiBoxHeight/10);
uiSignalOutPackingMode 	:= INT_TO_BYTE(uiPackingModeNo);

END_PROGRAM

// ---- POUs/P_Mqtt.TcPOU
PROGRAM P_Mqtt
VAR
  
	sCounter  : STRING(1024);
   
  	// Function blocks for IOT communication 
  	fbMqttClient    : FB_IotMqttClient;
	fbMessageQueue  : FB_IotMqttMessageQueue;
	fbMessage       : FB_IotMqttMessage;	
  
	bSetParameter   : BOOL := TRUE;  // set parametre 
	bHaveNetwork     : BOOL ; 
	
	(* publish message -  *)
	sTopicPub       	: STRING(255);
	sOpStateTopicPub	: STRING(255);
	sPLCStateTopicPub 	: STRING(255);
	sCutStateTopicPub	: STRING(255);
	sPickStateTopicPub	: STRING(255);
	sRecipeTopicPub		: STRING(255);
	sVelocityTopicPub	: STRING(255);
	sProgramTopicPub	: STRING(255);
	sAlarmTopicPub		: STRING(255);
	
	sPayloadPub     : STRING(255);
	
	bSendMsg         : BOOL;
	
	(* subscription *)
	bSubscribed     : BOOL;
	sTopicSub       : STRING(255);
	
	
	
	(* received message *)
	{attribute 'TcEncoding':='UTF-8'}
	sTopicRcv       : STRING(255);
	{attribute 'TcEncoding':='UTF-8'}
	sPayloadRcv     : STRING(255);
	bError           : BOOL;
	// Sent messages 
	udiSentMessages: UDINT;
	bstatus: BOOL;
	
	fbAdapterInfo: FB_GetAdaptersInfo;
	
	udiCounter : UDINT;
	
	tonSendMsg : Tc2_Standard.TON;
	
	tonMomOn : Tc2_Standard.TON;
	
	sTag : STRING;
	
	iFlag : INT;
	
	bCount : BOOL;
	bForceUpdate : BOOL;
	
END_VAR



 
  A_Init();

  // Connect Action 
  A_Connect();
  
  
  // Send Message Action
  A_SendMessage();
  
  // Subscribe Action
  A_Subscribe();
  
  // Get Adapter Info
  A_AdapterInfo();

ACTION A_AdapterInfo:

fbAdapterInfo(
	sNetID:='' , 
	bExecute:= NOT fbAdapterInfo.bExecute AND NOT fbAdapterInfo.bBusy , 
	tTimeout:= , 
	bBusy=> , 
	bError=> , 
	nErrID=> , 
	arrAdapters=> , 
	nCount=> , 
	nGet=> );
	
IF NOT fbAdapterInfo.bBusy THEN
	IF fbAdapterInfo.arrAdapters[0].sIpAddr <> '0.0.0.0' THEN
		bHaveNetwork:=TRUE;
	ELSE
		bHaveNetwork:=FALSE;
	END_IF
END_IF
END_ACTION

ACTION A_Connect:

// Execute and update MQTT client

fbMqttClient.Execute(bHaveNetwork);
bError:= fbMqttClient.bError;
END_ACTION

ACTION A_Init:

IF bSetParameter THEN

	fbMqttClient.sHostName:='192.168.29.56';
	fbMqttClient.nHostPort:=1883;
	
	fbMqttClient.nKeepAlive := 60;

	fbMqttClient.ipMessageQueue := fbMessageQueue;
		
	bSetParameter  := FALSE;
	
	sTopicPub 			:= 'mqtt/plc2hmi';
	sOpStateTopicPub	:= 'mqtt/plc2hmi/opState';
	sPLCStateTopicPub	:= 'mqtt/plc2hmi/plcState';
	sCutStateTopicPub	:= 'mqtt/plc2hmi/cutState';
	sPickStateTopicPub	:= 'mqtt/plc2hmi/pickState';
	sRecipeTopicPub		:= 'mqtt/plc2hmi/recipe';
	sVelocityTopicPub 	:= 'mqtt/plc2hmi/velocity';
	sProgramTopicPub 	:= 'mqtt/plc2hmi/program';
	sAlarmTopicPub 		:= 'mqtt/plc2hmi/alarm';
	
	sTopicSub 			:= 'php-mqtt/hmi2plc/#';
	
ELSIF NOT bHaveNetwork THEN
	bHaveNetwork := FALSE;

END_IF
END_ACTION

ACTION A_SendMessage:
// Send MQTT data 
IF fbMqttClient.bConnected AND bHaveNetwork THEN

	IF PROGRAM_DATA.usiRecipe <> PROGRAM_DATA.usiNewRecipe THEN
		///////////////////////////// RECIPE UPDATE //////////////////////////////
		PROGRAM_DATA.usiRecipe := PROGRAM_DATA.usiNewRecipe;
		sPayloadPub := USINT_TO_STRING(PROGRAM_DATA.usiRecipe);
		bstatus := fbMqttClient.Publish(sTopic:= sRecipeTopicPub, pPayload:= ADR(sPayloadPub), nPayloadSize:= LEN2(ADR(sPayloadPub)), eQoS:= TcIotMqttQos.AtMostOnceDelivery, bRetain:= TRUE, bQueue:= TRUE );
		udiSentMessages := udiSentMessages + 1; 
	END_IF

	IF bPLCStatus <> NewbPLCStatus OR bRobotCutStatus <> NewbRobotCutStatus OR bRobotPickStatus <> NewbRobotPickStatus THEN
		bPLCStatus 			:= NewbPLCStatus;
		bRobotCutStatus		:= NewbRobotCutStatus;
		bRobotPickStatus	:= NewbRobotPickStatus;
		
		// Onchange, publish PLC/Cut/Pick State
		sPayloadPub := BOOL_TO_STRING(bPLCStatus);
		bstatus := fbMqttClient.Publish(sTopic:= sPLCStateTopicPub, pPayload:= ADR(sPayloadPub), nPayloadSize:= LEN2(ADR(sPayloadPub)), eQoS:= TcIotMqttQos.AtMostOnceDelivery, bRetain:= TRUE, bQueue:= TRUE );
		udiSentMessages := udiSentMessages + 1; 
		
		sPayloadPub := BOOL_TO_STRING(bRobotCutStatus);
		bstatus := fbMqttClient.Publish(sTopic:= sCutStateTopicPub, pPayload:= ADR(sPayloadPub), nPayloadSize:= LEN2(ADR(sPayloadPub)), eQoS:= TcIotMqttQos.AtMostOnceDelivery, bRetain:= TRUE, bQueue:= TRUE );
		udiSentMessages := udiSentMessages + 1; 
		
		sPayloadPub := BOOL_TO_STRING(bRobotPickStatus);
		bstatus := fbMqttClient.Publish(sTopic:= sPickStateTopicPub, pPayload:= ADR(sPayloadPub), nPayloadSize:= LEN2(ADR(sPayloadPub)), eQoS:= TcIotMqttQos.AtMostOnceDelivery, bRetain:= TRUE, bQueue:= TRUE );
		udiSentMessages := udiSentMessages + 1; 
	END_IF

	////////////////////////////////// MAIN page HMI ////////////////////////////////////
	(*IF PROGRAM_DATA.usiProgram <> PROGRAM_DATA.usiNewProgram THEN*)
	IF PROGRAM_DATA.usiNewProgram <> 0 THEN
		PROGRAM_DATA.usiProgram := PROGRAM_DATA.usiNewProgram;
		
		sPayloadPub := USINT_TO_STRING(PROGRAM_DATA.usiProgram);
		bstatus := fbMqttClient.Publish(sTopic:= sProgramTopicPub, pPayload:= ADR(sPayloadPub), nPayloadSize:= LEN2(ADR(sPayloadPub)), eQoS:= TcIotMqttQos.AtMostOnceDelivery, bRetain:= TRUE, bQueue:= TRUE );
		(*udiSentMessages := udiSentMessages + 1; *)
	END_IF
	
	IF PROGRAM_DATA.usiVelocity <> PROGRAM_DATA.usiNewVelocity THEN
		PROGRAM_DATA.usiVelocity := PROGRAM_DATA.usiNewVelocity;
		
		sPayloadPub := USINT_TO_STRING(PROGRAM_DATA.usiVelocity);
		bstatus := fbMqttClient.Publish(sTopic:= sVelocityTopicPub, pPayload:= ADR(sPayloadPub), nPayloadSize:= LEN2(ADR(sPayloadPub)), eQoS:= TcIotMqttQos.AtMostOnceDelivery, bRetain:= TRUE, bQueue:= TRUE );
		udiSentMessages := udiSentMessages + 1; 
	END_IF
	
	IF bStart AND iFlag <> 1 THEN
		iFlag := 1;
		// When running, publish start
		sPayloadPub := 'start';
		bstatus := fbMqttClient.Publish(sTopic:= sOpStateTopicPub, pPayload:= ADR(sPayloadPub), nPayloadSize:= LEN2(ADR(sPayloadPub)), eQoS:= TcIotMqttQos.AtMostOnceDelivery, bRetain:= TRUE, bQueue:= TRUE );
		udiSentMessages := udiSentMessages + 1; 
	ELSIF ((bStop) OR (gStopped = TRUE)) AND iFlag <> 2 THEN
		iFlag := 2;
		// When stopped, publish stop
		sPayloadPub := 'stop';
		bstatus := fbMqttClient.Publish(sTopic:= sOpStateTopicPub, pPayload:= ADR(sPayloadPub), nPayloadSize:= LEN2(ADR(sPayloadPub)), eQoS:= TcIotMqttQos.AtMostOnceDelivery, bRetain:= TRUE, bQueue:= TRUE );
		udiSentMessages := udiSentMessages + 1; 
	ELSIF (bAlarm OR bAlarmAck) AND iFlag <> 3 THEN
		iFlag := 3;
		sPayloadPub := TO_STRING(robotAlarmId);
		bstatus := fbMqttClient.Publish(sTopic:= sAlarmTopicPub, pPayload:= ADR(sPayloadPub), nPayloadSize:= LEN2(ADR(sPayloadPub)), eQoS:= TcIotMqttQos.AtMostOnceDelivery, bRetain:= TRUE, bQueue:= TRUE );
		udiSentMessages := udiSentMessages + 1; 
	END_IF
	


	IF bSendMsg AND iFlag <> 3 THEN // Send data
		iFlag := 3;
		bSendMsg := FALSE;
		 // Publish method - send payload       
		bstatus := fbMqttClient.Publish(sTopic:= sTopicPub, pPayload:= ADR(sCounter), nPayloadSize:= LEN2(ADR(sCounter)), eQoS:= TcIotMqttQos.AtMostOnceDelivery, bRetain:= FALSE, bQueue:= FALSE );
	  udiSentMessages := udiSentMessages + 1; 
 	END_IF
END_IF
END_ACTION

ACTION A_Subscribe:



// Subscribe (modtage) messages with a connection to AZURE is established
IF fbMqttClient.bConnected THEN
  // Subscribe only if not already subscriped
	IF NOT bSubscribed THEN
    // Call of subscribe Method
		bSubscribed := fbMqttClient.Subscribe(sTopic:=sTopicSub, eQoS:=TcIotMqttQos.AtLeastOnceDelivery);
	END_IF
ELSE
	bSubscribed := FALSE;
END_IF




//Get messages with the use of a queue system
IF fbMessageQueue.nQueuedMessages > 0 THEN
	IF fbMessageQueue.Dequeue(fbMessage:=fbMessage) THEN
		fbMessage.GetTopic(pTopic:=ADR(sTopicRcv), nTopicSize:=SIZEOF(sTopicRcv) );
		fbMessage.GetPayload(pPayload:=ADR(sPayloadRcv), nPayloadSize:=SIZEOF(sPayloadRcv), bSetNullTermination:=TRUE);
		
		sTag := MID(STR:= sTopicRcv, LEN:= Tc2_Standard.LEN(sTopicRcv)-12, POS:= 13);		
		
		IF sTopicRcv = 'php-mqtt/hmi2plc/recipe' THEN
			PROGRAM_DATA.usiNewRecipe := STRING_TO_USINT(sPayloadRcv);
			P_SqlSelectRecipe.bRead := TRUE;
		END_IF
		
		IF sTopicRcv = 'php-mqtt/hmi2plc/program' THEN
			PROGRAM_DATA.usiNewProgram := STRING_TO_USINT(sPayloadRcv);
			//P_SqlSelectRecipe.bRead := TRUE;
		END_IF
		
		IF sTopicRcv = 'php-mqtt/hmi2plc/setup' THEN
			IF (sPayloadRcv = 'rob-con') THEN
				bRobotConnect 		:= TRUE;
			ELSIF (sPayloadRcv = 'rob-discon') THEN 	
				bRobotDisconnect	:= TRUE;
			ELSIF (sPayloadRcv = 'calib-check') THEN 	
				bCalibCheck 		:= TRUE;
			END_IF
		END_IF
		
		IF sTopicRcv = 'php-mqtt/hmi2plc/calib' THEN
			sNewCalib := sPayloadRcv;
		END_IF
		
		IF sTopicRcv = 'php-mqtt/hmi2plc/vision' THEN
			usiVisionCmd := STRING_TO_USINT(sPayloadRcv);
		END_IF
		
		IF sTopicRcv = 'php-mqtt/hmi2plc/tool' THEN
			sToolControl := sPayloadRcv;
		END_IF
		
		IF sTopicRcv = 'php-mqtt/hmi2plc/frameUpdate' THEN
			P_SqlSelectFrame.bRead := TRUE;
		END_IF
		
		IF sTopicRcv = 'php-mqtt/hmi2plc/frameUpdate' THEN
			P_SqlSelectFrame.bRead := TRUE;
		END_IF
		
		IF sTopicRcv = 'php-mqtt/hmi2plc/alarm' THEN
			IF (sPayloadRcv = 'Acknowledge') THEN
				bAlarm := FALSE;
			END_IF
		END_IF
		
		IF sTopicRcv = 'php-mqtt/hmi2plc/opState' THEN
			IF (sPayloadRcv = 'start') THEN
				bStart	:= TRUE;
				bStop 	:= FALSE;
			ELSIF (sPayloadRcv = 'pause') THEN
				bStop 	:= TRUE;
				bStart	:= FALSE;
			ELSIF (sPayloadRcv = 'stop') THEN
				bStop := TRUE;
				bStart	:= FALSE;
			END_IF
		END_IF
		
		IF	sPayloadRcv = '1' THEN
			IF sTopicRcv = 'php-mqtt/hmi2plc/resetWith' THEN
				bResetButton := TRUE;
			ELSIF sTopicRcv = 'php-mqtt/hmi2plc/resetWithout' THEN
				bResetButton2 := TRUE;
			ELSIF sTopicRcv = 'php-mqtt/hmi2plc/serviceStart' THEN
				bRobotServiceStart := TRUE;
			ELSIF sTopicRcv = 'php-mqtt/hmi2plc/serviceStop' THEN
				bRobotServiceStop := TRUE;
			ELSIF sTopicRcv = 'php-mqtt/hmi2plc/idle' THEN
				bBackToZero := TRUE;
			END_IF
		END_IF
			
		IF sPayloadRcv = '0' THEN
			IF sTopicRcv = 'php-mqtt/hmi2plc/resetWith' THEN
				bResetButton := FALSE;
			ELSIF sTopicRcv = 'php-mqtt/hmi2plc/resetWithout' THEN
				bResetButton2 := FALSE;
			ELSIF sTopicRcv = 'php-mqtt/hmi2plc/serviceStart' THEN
				bRobotServiceStart := FALSE;
			ELSIF sTopicRcv = 'php-mqtt/hmi2plc/serviceStop' THEN
				bRobotServiceStop := FALSE;
			ELSIF sTopicRcv = 'php-mqtt/hmi2plc/idle' THEN
				bBackToZero := FALSE;
			END_IF
			
		END_IF
			
		
		
		IF sTag = 'reset' THEN
			udiCounter := 0;
			bForceUpdate := TRUE;
		ELSIF sTag = 'start' THEN	
			bCount := TO_BOOL(sPayloadRcv);
		END_IF
		
	END_IF
END_IF

tonMomOn(PT:= T#100MS, Q=> , ET=> );
END_ACTION

END_PROGRAM

// ---- POUs/SQL/03_Select/P_SqlSelectRecipe.TcPOU
PROGRAM P_SqlSelectRecipe
VAR_INPUT
	bRead : BOOL; //Execute command
END_VAR
VAR
	
	fbSq : FB_EasySql;
	sSql : STRING(1000);
	
	iGE : INT:=1; //Select value
	
	astData : ARRAY[0..9] OF ST_SelectRecipeStruct; //Data array for recieved data
	
	bDone : BOOL; //Command done
	bError : BOOL; //Command error
	sError : STRING(255);
	
	udiNoOfRecords : UDINT; //Numbers of returned recoreds
	
END_VAR

//Select data from database
sSql := 'SELECT * from tpr_db.recipe WHERE recipe_id =¤1¤';

F_Replace(pString:= ADR(sSql), cbStringLen:= SIZEOF(sSql), sSearch:= '¤1¤', sReplace:= TO_STRING(PROGRAM_DATA.usiRecipe)); //Replace placeholder

fbSq(
	bExecute:= bRead, 
	wDBID:= 1, 
	pSql:= ADR(sSql), 
	cbSql:= SIZEOF(sSql), 
	pData:= ADR(astData), 
	cbData:= SIZEOF(astData), 
	udiMaxOfRecord:= 3, //Max number of recieved records
	udiNoOfRecords=> udiNoOfRecords, 
	bDone=> bDone, 
	bBusy=> , 
	bError=> bError, 
	sError=> sError
);

END_PROGRAM

// ---- POUs/EasySql/F_FB/FB_EasySql.TcPOU
//------------------------------------------------------------------------------------------
//                                                                                        	
//***************************** Beckhoff TwinCAT Examples **********************************
//                                                                                        	
//************************************* WARNING ********************************************
// This program is only an example. If it is used as a control program in any real        	
// application, Beckhoff is not responsible for any malfunction, loss or damage           	
// which could arise by using this program!                                               	
//                                                                                        	
//*************************************  Program Info. *************************************
//                                                                                        	
// PLC program name:       	F_Replace (Function)               	                           	
// Software platform:      	TwinCat v3.1.4024.10
//							Database Server 3.3.33.1				                          	
// Modified by:            	Per Søgaard Carlsen 			                                  	
// Email:					p.carlsen@beckhoff.com	                                  	
//                                                                                        	
// ======================================================================================== 
//         Version       Date                        Remarks                              	
// ======================================================================================== 
//         1.0           10 july 2020                 First release of this example        	
// ======================================================================================== 
//                                                                                        	
//******************************* Aims OF this PLC PROGRAM *********************************
//                                                                                        	
// Execute SQL quires in expert mode						 			                             
//                                                                                        	
//-----------------------------------------------------------------------------------------

FUNCTION_BLOCK FB_EasySql

VAR_INPUT
	bExecute : BOOL;
	wDBID : WORD; //DBID
	pSql : POINTER TO BYTE; //Pointer to SQL command string
	cbSql : UDINT; //Sizeof of SSql command string
	pData : POINTER TO BYTE; //Pointer to data array to store readed data from database - set to 0 for write
	cbData : UDINT; //Sizeof data array for stored data.  - set to 0 for write
	udiMaxOfRecord : UDINT; //Maximum numbers of data record to read.
END_VAR
	
VAR_OUTPUT
	udiNoOfRecords : UDINT; //Hvor mange record er fundet
	bDone : BOOL; //Database skrivning afsluttet
	bBusy : BOOL; //Database skrivning afsluttet
	bError : BOOL; //Fejl under skrivning til database
	sError : STRING(255); //Fejl beskrivelse
END_VAR

VAR
	fbSqlConnection : FB_SQLDatabaseEvt(sNetID:='',tTimeout:=T#5S);
	fbSqlCommand : FB_SQLCommandEvt(sNetID:='',tTimeout:=T#5S);
	fbSqlResult : FB_SQLResultEvt(sNetID:='', tTimeout   := T#5S);
	iState : INT;
	ipResultEvent : Tc3_Eventlogger.I_TcMessage;
	bInternDone : BOOL;
	bInternError : BOOL;
END_VAR

CASE iState OF
	0:
		
		IF bExecute THEN //Whait for start
			bBusy := TRUE;
			M_Zero();
			iState := 100;
		END_IF
					
	100: //Open database connection

		fbSqlConnection.Connect(hDBID:= wDBID);
				
		IF NOT fbSqlConnection.bBusy THEN
			IF fbSqlConnection.bError THEN
				ipResultEvent := fbSqlConnection.ipTcResult;
				iState := 9000;	
			ELSE
				iState := 110;	
			END_IF
		END_IF
				
	110: //Init SQL command
											
		IF fbSqlConnection.CreateCmd(ADR(fbSqlCommand)) THEN
			IF fbSqlConnection.bError THEN
				ipResultEvent := fbSqlConnection.ipTcResult;
				iState := 9000;
			ELSE
				IF pData = 0 OR cbData = 0 OR udiMaxOfRecord = 0 THEN
					iState := 130;	
				ELSE
					iState := 120;
				END_IF
				
			END_IF
		END_IF		
				
	120: //Execute SQL command, with data return
			
		IF fbSqlCommand.ExecuteDataReturn(pSQLCmd:=pSql , cbSQLCmd:= cbSql, pSQLDBResult:= ADR(fbSQLResult)) THEN
			ipResultEvent := fbSqlCommand.ipTcResult;
				
			IF udiMaxOfRecord < 1 THEN // Minimum read one record
				udiMaxOfRecord := 1;
			END_IF
					
						
			IF fbSqlResult.Read(0, udiMaxOfRecord, pData, cbData, TRUE, TRUE) THEN //Parse sql data to struct
				IF fbSqlResult.bError THEN
					ipResultEvent := fbSqlResult.ipTcResult;
					udiNoOfRecords := 0;
					iState := 9000; 
				ELSE
					// Data found without any errors
					udiNoOfRecords := fbSqlResult.nDataCount; 
					bInternDone := TRUE;
					iState := 1000; 
				END_IF
			END_IF
			
		END_IF
		
	130: //Execute SQL command, without data return
		IF fbSqlCommand.Execute(pSQLCmd:= pSql, cbSQLCmd:= cbSql) THEN
			IF fbSqlCommand.bError THEN
				ipResultEvent := fbSqlCommand.ipTcResult;
				udiNoOfRecords := 0;
				iState := 9000; 
			ELSE
				// Write data without any errors
				udiNoOfRecords := fbSqlResult.nDataCount; 
				bInternDone := TRUE;
				iState := 1000; 
			END_IF
		END_IF
				
	1000: //Close database connection
		fbSqlConnection.Disconnect();	
		IF NOT fbSqlConnection.bBusy THEN
			iState := 1010;
		END_IF
			
	1010: // Return to start
		bBusy := FALSE;
		bDone := bInternDone;
		bError := bInternError;
		IF NOT bExecute THEN
			bDone := FALSE;
			iState := 0;
		END_IF
								
	9000: //Parse error description
		bInternError := TRUE;
		IF ipResultEvent.RequestEventText(nLangId:= 1033, sResult:= sError, nResultSize:= SIZEOF(sError), bError=> , hrErrorCode=> ) THEN
			iState := 1000;
		END_IF
	
END_CASE

METHOD PRIVATE M_Zero : BOOL
VAR_INPUT
END_VAR
sError := '';
bBusy := FALSE;
bError := FALSE;
bInternError := FALSE;
bDone := FALSE;
bInternDone := FALSE;
udiNoOfRecords := 0;
END_METHOD

END_FUNCTION_BLOCK

// ---- POUs/EasySql/F_FB/F_Replace.TcPOU
//------------------------------------------------------------------------------------------
//                                                                                        	
//***************************** Beckhoff TwinCAT Examples **********************************
//                                                                                        	
//************************************* WARNING ********************************************
// This program is only an example. If it is used as a control program in any real        	
// application, Beckhoff is not responsible for any malfunction, loss or damage           	
// which could arise by using this program!                                               	
//                                                                                        	
//*************************************  Program Info. *************************************
//                                                                                        	
// PLC program name:       	F_Replace (Function)               	                           	
// Software platform:      	TwinCat v3.1.4024.10				                          	
// Modified by:            	Per Søgaard Carlsen 			                                  	
// Email:					p.carlsen@beckhoff.com	                                  	
//                                                                                        	
// ======================================================================================== 
//         Version       Date                        Remarks                              	
// ======================================================================================== 
//         1.0           10 july 2020                 First release of this example        	
// ======================================================================================== 
//                                                                                        	
//******************************* Aims OF this PLC PROGRAM *********************************
//                                                                                        	
// Compleate search and replace function in long strings						 			                             
//                                                                                        	
//-----------------------------------------------------------------------------------------
FUNCTION F_Replace : bool
VAR_INPUT
	pString : POINTER TO STRING; //Pointer to source and destination string.
	cbStringLen : UDINT; //Lenght of source and destination string
	sSearch : STRING(255); //Search in string
	sReplace : STRING(255); //Releace in string
END_VAR
VAR
	udiStartPos : UDINT; //Start position for found search result
	udiFindPos : UDINT; //Search start position in string
	bFoundOne : BOOL; //One ore more replace done
	bFoundThis : BOOL;
END_VAR

bFoundOne := FALSE; //Min one item replaced
udiFindPos := 0; //Search from position in string

REPEAT
	bFoundThis := FALSE;
	udiStartPos := udiFindPos;
	
	IF 	udiFindPos <= LEN2(pSTRING:= pString) THEN
		//Search
		udiFindPos := FIND2(pSrcString:= pString+udiStartPos, pFindString:= ADR(sSearch));
	ELSE
		//No match found
		udiFindPos := 0;
	END_IF
	
	IF udiFindPos <> 0 THEN
		//Replace item
		REPLACE2(
		pSrcString:= pString+udiStartPos, 
		pInsertString:= ADR(sReplace), 
		pDstString:= pString, 
		nDstSize:= cbStringLen-udiStartPos, 
		nLen:= Tc2_Utilities.LEN2(ADR(sSearch)), 
		nPos:= udiFindPos);
		bFoundOne := TRUE;
		bFoundThis := TRUE;	
		
		udiFindPos := udiFindPos + TO_UDINT(Tc2_Standard.LEN(sReplace)); //Update search from position
		
		
	END_IF
	
	UNTIL NOT bFoundThis //Repeat until all item found and replaced
END_REPEAT

F_Replace := bFoundOne;

END_FUNCTION

// ---- POUs/SQL/03_Select/P_SqlSelectFrame.TcPOU
PROGRAM P_SqlSelectFrame
VAR_INPUT
	bRead : BOOL; //Execute command
END_VAR
VAR
	
	fbSq : FB_EasySql;
	sSql : STRING(1000);
	
	iGE : INT:=1; //Select value
	
	astData : ARRAY[0..9] OF ST_SelectFrameStruct; //Data array for recieved data
	
	bDone : BOOL; //Command done
	bError : BOOL; //Command error
	sError : STRING(255);
	
	udiNoOfRecords : UDINT; //Numbers of returned recoreds
	
END_VAR

//Select data from database
sSql := 'SELECT * from frame';

F_Replace(pString:= ADR(sSql), cbStringLen:= SIZEOF(sSql), sSearch:= '¤1¤', sReplace:= TO_STRING(PROGRAM_DATA.usiRecipe)); //Replace placeholder

fbSq(
	bExecute:= bRead, 
	wDBID:= 1, 
	pSql:= ADR(sSql), 
	cbSql:= SIZEOF(sSql), 
	pData:= ADR(astData), 
	cbData:= SIZEOF(astData), 
	udiMaxOfRecord:= 3, //Max number of recieved records
	udiNoOfRecords=> udiNoOfRecords, 
	bDone=> bDone, 
	bBusy=> , 
	bError=> bError, 
	sError=> sError
);

END_PROGRAM

// ---- POUs/SQL/00_TestData/P_SqlGeneratTestData.TcPOU
PROGRAM P_SqlGeneratTestData
VAR
	
	fbSql : FB_EasySql;
	sSql : STRING(1000);
	sSqlInser : STRING(1000):='INSERT INTO myTable (myId,myCustomer,myValue) VALUES (1,$'Martin$',1.1),(2,$'Hans$',2.2),(3,$'Bjarne$',3.3),(4,$'Niels$',4.4),(5,$'Bo$',5.5),(6,$'Allan$',6.6),(7,$'Tom$',7.7),(8,$'Tom$',8.8),(9,$'Tom$',9.9),(10,$'Kurt$',10.1),(11,$'Kurt$',11.11)';	
		
	bDone : BOOL; //Command done
	bError : BOOL; //Command error
	sError : STRING(255);
	
	bStart : BOOL;
	iState : INT;
	
	
END_VAR

//Clean database and inserty test items.
CASE iState OF
	0:
		fbSql.pData := 0;
		fbSql.cbData := 0;
		fbSql.cbData := 0;
		fbSql.bExecute := FALSE;
		iState := 10;
		
	10:
		IF bStart THEN
			bStart := FALSE;
			iState := 100;
		END_IF
		
	100: // Truncate database
		sSql := 'DELETE FROM myTable'; //Normaly use TRUNCATE - but SqLite dont support TRUNCATE
		fbSql.pData := 0;
		fbSql.cbData := 0;
		fbSql.cbData := 0;
		fbSql.bExecute := TRUE;
		iState := 110;
		
	110:
		IF fbSql.bDone THEN
			fbSql.bExecute := FALSE;
			iState := 120;
		END_IF
		
	120:
		sSql := 'VACUUM'; //Normaly use TRUNCATE - but SqLite dont support TRUNCATE
		fbSql.bExecute := TRUE;
		iState := 130;
		
	130:
		IF NOT fbSql.bDone THEN
			fbSql.bExecute := FALSE;
			iState := 140;
		END_IF
		
	140:
		sSql := sSqlInser;
		fbSql.bExecute := TRUE;
		iState := 150;
		
	150:
		IF fbSql.bDone THEN
			iState := 0;
		END_IF
		


END_CASE



fbSql(
	bExecute:= , 
	wDBID:= 1, 
	pSql:= ADR(sSql), 
	cbSql:= SIZEOF(sSql), 
	pData:= , 
	cbData:= , 
	udiMaxOfRecord:= 0, 
	udiNoOfRecords=> , 
	bDone=> bDone, 
	bBusy=> , 
	bError=> bError, 
	sError=> sError);

END_PROGRAM

// ---- POUs/SQL/03_Select/P_SqlSelect.TcPOU
PROGRAM P_SqlSelect
VAR
	
	fbSq : FB_EasySql;
	sSql : STRING(1000);
	
	iGE : INT:=1; //Select value
	
	astData : ARRAY[0..9] OF ST_SelectStruct; //Data array for recieved data
	
	bRead : BOOL; //Execute command
	bDone : BOOL; //Command done
	bError : BOOL; //Command error
	sError : STRING(255);
	
	udiNoOfRecords : UDINT; //Numbers of returned recoreds
	
END_VAR

//Select data from database
sSql := 'SELECT id,username,password FROM tpr_db.user where id >=¤1¤';

F_Replace(pString:= ADR(sSql), cbStringLen:= SIZEOF(sSql), sSearch:= '¤1¤', sReplace:= TO_STRING(iGE)); //Replace placeholder

fbSq(
	bExecute:= bRead, 
	wDBID:= 1, 
	pSql:= ADR(sSql), 
	cbSql:= SIZEOF(sSql), 
	pData:= ADR(astData), 
	cbData:= SIZEOF(astData), 
	udiMaxOfRecord:= 3, //Max number of recieved records
	udiNoOfRecords=> udiNoOfRecords, 
	bDone=> bDone, 
	bBusy=> , 
	bError=> bError, 
	sError=> sError
);

END_PROGRAM

// ---- POUs/SQL/03_Select/P_SqlSelectCurrent.TcPOU
PROGRAM P_SqlSelectCurrent
VAR_INPUT
	bRead : BOOL; //Execute command
END_VAR
VAR
	
	fbSq : FB_EasySql;
	sSql : STRING(1000);
	
	iGE : INT:=1; //Select value
	
	astData : ARRAY[0..9] OF ST_SelectCurrentStruct; //Data array for recieved data
	
	bDone : BOOL; //Command done
	bError : BOOL; //Command error
	sError : STRING(255);
	
	udiNoOfRecords : UDINT; //Numbers of returned recoreds
	
END_VAR

//Select data from database
sSql := 'SELECT * from tpr_db.currentValues';

//F_Replace(pString:= ADR(sSql), cbStringLen:= SIZEOF(sSql), sSearch:= '¤1¤', sReplace:= TO_STRING(PROGRAM_DATA.usiRecipe)); //Replace placeholder

fbSq(
	bExecute:= bRead, 
	wDBID:= 1, 
	pSql:= ADR(sSql), 
	cbSql:= SIZEOF(sSql), 
	pData:= ADR(astData), 
	cbData:= SIZEOF(astData), 
	udiMaxOfRecord:= 3, //Max number of recieved records
	udiNoOfRecords=> udiNoOfRecords, 
	bDone=> bDone, 
	bBusy=> , 
	bError=> bError, 
	sError=> sError
);

END_PROGRAM

// ---- POUs/SQL/03_Select/P_SqlSelectAlarm.TcPOU
PROGRAM P_SqlSelectAlarm
VAR_INPUT
	bRead : BOOL; //Execute command
END_VAR
VAR
	
	fbSq : FB_EasySql;
	sSql : STRING(1000);
	
	iGE : INT:=1; //Select value
	
	astData : ARRAY[0..9] OF ST_SelectAlarmStruct; //Data array for recieved data
	
	bDone : BOOL; //Command done
	bError : BOOL; //Command error
	sError : STRING(255);
	
	udiNoOfRecords : UDINT; //Numbers of returned recoreds
	
END_VAR

//Select data from database
sSql := 'SELECT * from systemAlarms WHERE alarmId = ¤1¤;';

F_Replace(pString:= ADR(sSql), cbStringLen:= SIZEOF(sSql), sSearch:= '¤1¤', sReplace:= TO_STRING(robotAlarmId)); //Replace placeholder

fbSq(
	bExecute:= bRead, 
	wDBID:= 1, 
	pSql:= ADR(sSql), 
	cbSql:= SIZEOF(sSql), 
	pData:= ADR(astData), 
	cbData:= SIZEOF(astData), 
	udiMaxOfRecord:= 3, //Max number of recieved records
	udiNoOfRecords=> udiNoOfRecords, 
	bDone=> bDone, 
	bBusy=> , 
	bError=> bError, 
	sError=> sError
);

END_PROGRAM

// ---- POUs/SQL/03_Select/P_SqlSelectAlarmLog.TcPOU
PROGRAM P_SqlSelectAlarmLog
VAR_INPUT
	bRead : BOOL; //Execute command
END_VAR
VAR
	
	fbSq : FB_EasySql;
	sSql : STRING(1000);
	
	iGE : INT:=1; //Select value
	
	astData : ARRAY[0..9] OF ST_SelectAlarmLogStruct; //Data array for recieved data
	
	bDone : BOOL; //Command done
	bError : BOOL; //Command error
	sError : STRING(255);
	
	udiNoOfRecords : UDINT; //Numbers of returned recoreds
	
END_VAR

//Select data from database
sSql := 'SELECT * from alarmLog ORDER BY time DESC LIMIT 1;';

//F_Replace(pString:= ADR(sSql), cbStringLen:= SIZEOF(sSql), sSearch:= '¤1¤', sReplace:= TO_STRING(robotAlarmId)); //Replace placeholder

fbSq(
	bExecute:= bRead, 
	wDBID:= 1, 
	pSql:= ADR(sSql), 
	cbSql:= SIZEOF(sSql), 
	pData:= ADR(astData), 
	cbData:= SIZEOF(astData), 
	udiMaxOfRecord:= 3, //Max number of recieved records
	udiNoOfRecords=> udiNoOfRecords, 
	bDone=> bDone, 
	bBusy=> , 
	bError=> bError, 
	sError=> sError
);

END_PROGRAM

// ---- POUs/SQL/03_Select/P_SqlSelectTop.TcPOU
PROGRAM P_SqlSelectTop
VAR
	
	fbSq : FB_EasySql;
	sSql : STRING(1000);
	
	iGE : INT:=1; //Select value
	
	astData : ARRAY[0..9] OF ST_SelectStruct; //Data array for recieved data
	
	bRead : BOOL; //Execute command
	bDone : BOOL; //Command done
	bError : BOOL; //Command error
	sError : STRING(255);
	
	udiNoOfRecords : UDINT; //Numbers of returned recoreds
	udiMaxOfRecord : UDINT;
	
END_VAR

//Select data from database, only return max numbers of records from Database to database server.
udiMaxOfRecord := 3;
sSql := 'SELECT myId,myCustomer,myValue FROM myTable where myId >¤1¤ ORDER BY myId LIMIT ¤2¤'; // Only transmit LIMIT numbers of record from database to TC Database server

F_Replace(pString:= ADR(sSql), cbStringLen:= SIZEOF(sSql), sSearch:= '¤1¤', sReplace:= TO_STRING(iGE)); //Replace placeholder
F_Replace(pString:= ADR(sSql), cbStringLen:= SIZEOF(sSql), sSearch:= '¤2¤', sReplace:= TO_STRING(udiMaxOfRecord)); //Replace placeholder

fbSq(
	bExecute:= bRead, 
	wDBID:= 1, 
	pSql:= ADR(sSql), 
	cbSql:= SIZEOF(sSql), 
	pData:= ADR(astData), 
	cbData:= SIZEOF(astData), 
	udiMaxOfRecord:= udiMaxOfRecord, //Max number of recieved records
	udiNoOfRecords=> udiNoOfRecords, 
	bDone=> bDone, 
	bBusy=> , 
	bError=> bError, 
	sError=> sError);

END_PROGRAM

// ---- POUs/SQL/01_Insert/P_SqlInsert.TcPOU
PROGRAM P_SqlInsert
VAR
	
	fbSql : FB_EasySql;
	sSql : STRING(1000);
		
	iId : INT; //Insert data
	sCustomer : STRING; //Insert data
	rValue : REAL; //Insert data
		
	bInsert : BOOL; //Execute command
	bDone : BOOL; //Command done
	bError : BOOL; //Command error
	sError : STRING(255);
	
END_VAR

// Insert new items to database
sSql := 'INSERT INTO tpr_db.test (test) VALUES (¤1¤)';

F_Replace(pString:= ADR(sSql), cbStringLen:= SIZEOF(sSql), sSearch:= '¤1¤', sReplace:= TO_STRING(123)); //Replace placeholder
//F_Replace(pString:= ADR(sSql), cbStringLen:= SIZEOF(sSql), sSearch:= '¤2¤', sReplace:= sCustomer); //Replace placeholder
//F_Replace(pString:= ADR(sSql), cbStringLen:= SIZEOF(sSql), sSearch:= '¤3¤', sReplace:= TO_STRING(rValue)); //Replace placeholder

fbSql(
	bExecute:= bInsert, 
	wDBID:= 1, 
	pSql:= ADR(sSql), 
	cbSql:= SIZEOF(sSql), 
	pData:= 0, 
	cbData:= 0, 
	udiMaxOfRecord:= 0, 
	udiNoOfRecords=> , 
	bDone=> bDone, 
	bBusy=> , 
	bError=> bError, 
	sError=> sError);

END_PROGRAM

// ---- POUs/SQL/01_Insert/P_SqlInsertAlarmLog.TcPOU
PROGRAM P_SqlInsertAlarmLog
VAR_INPUT
	bInsert : BOOL; //Execute command
END_VAR
VAR
	
	fbSql : FB_EasySql;
	sSql : STRING(1000);
		
	iId : INT; //Insert data
	sCustomer : STRING; //Insert data
	rValue : REAL; //Insert data
		
	
	bDone : BOOL; //Command done
	bError : BOOL; //Command error
	sError : STRING(255);
	
END_VAR

// Insert new items to database
sSql := 'INSERT INTO tpr_db.alarmLog (alarmId, deviceWhich) VALUES (¤1¤, "¤2¤");';

F_Replace(pString:= ADR(sSql), cbStringLen:= SIZEOF(sSql), sSearch:= '¤1¤', sReplace:= TO_STRING(robotAlarmId)); //Replace placeholder
F_Replace(pString:= ADR(sSql), cbStringLen:= SIZEOF(sSql), sSearch:= '¤2¤', sReplace:= TO_STRING(sDeviceWhich)); //Replace placeholder
//F_Replace(pString:= ADR(sSql), cbStringLen:= SIZEOF(sSql), sSearch:= '¤3¤', sReplace:= TO_STRING(rValue)); //Replace placeholder

fbSql(
	bExecute:= bInsert, 
	wDBID:= 1, 
	pSql:= ADR(sSql), 
	cbSql:= SIZEOF(sSql), 
	pData:= 0, 
	cbData:= 0, 
	udiMaxOfRecord:= 0, 
	udiNoOfRecords=> , 
	bDone=> bDone, 
	bBusy=> , 
	bError=> bError, 
	sError=> sError);

END_PROGRAM

// ---- POUs/SQL/01_Insert/P_SqlInsertLog.TcPOU
PROGRAM P_SqlInsertLog
VAR_INPUT
	bInsert : BOOL; //Execute command
END_VAR
VAR
	
	fbSql : FB_EasySql;
	sSql : STRING(1000);
		
	iId : INT; //Insert data
	sCustomer : STRING; //Insert data
	rValue : REAL; //Insert data
		
	
	bDone : BOOL; //Command done
	bError : BOOL; //Command error
	sError : STRING(255);
	
END_VAR

// Insert new items to database
sSql := 'INSERT INTO tpr_db.log (runTime, imageAmount, stickoutCut, retry, imgCnfgChange, success) VALUES (¤1¤, ¤2¤, ¤3¤, ¤4¤, ¤5¤, ¤6¤);';

F_Replace(pString:= ADR(sSql), cbStringLen:= SIZEOF(sSql), sSearch:= '¤1¤', sReplace:= TO_STRING(uiElapsedTime)); //Replace placeholder
F_Replace(pString:= ADR(sSql), cbStringLen:= SIZEOF(sSql), sSearch:= '¤2¤', sReplace:= TO_STRING(usiImageLog)); //Replace placeholder
F_Replace(pString:= ADR(sSql), cbStringLen:= SIZEOF(sSql), sSearch:= '¤3¤', sReplace:= TO_STRING(usiStickoutCutLog)); //Replace placeholder
F_Replace(pString:= ADR(sSql), cbStringLen:= SIZEOF(sSql), sSearch:= '¤4¤', sReplace:= TO_STRING(usiRetryLog)); //Replace placeholder
F_Replace(pString:= ADR(sSql), cbStringLen:= SIZEOF(sSql), sSearch:= '¤5¤', sReplace:= TO_STRING(usiImageRetry)); //Replace placeholder
F_Replace(pString:= ADR(sSql), cbStringLen:= SIZEOF(sSql), sSearch:= '¤6¤', sReplace:= TO_STRING(bLogSucces)); //Replace placeholder

fbSql(
	bExecute:= bInsert, 
	wDBID:= 1, 
	pSql:= ADR(sSql), 
	cbSql:= SIZEOF(sSql), 
	pData:= 0, 
	cbData:= 0, 
	udiMaxOfRecord:= 0, 
	udiNoOfRecords=> , 
	bDone=> bDone, 
	bBusy=> , 
	bError=> bError, 
	sError=> sError);

END_PROGRAM

// ---- POUs/SQL/01_Insert/P_SqlInsertRowConstructor.TcPOU
PROGRAM P_SqlInsertRowConstructor
VAR
	
	fbSql : FB_EasySql;
	sSql : STRING(1000);
		
	aiId : ARRAY[0..1] OF INT; //Insert data
	asCustomer : ARRAY[0..1] OF STRING; //Insert data
	arValue : ARRAY[0..1] OF REAL; //Insert data
		
	bInsert : BOOL; //Execute command
	bDone : BOOL; //Command done
	bError : BOOL; //Command error
	sError : STRING(255);
	
END_VAR

// Insert more than one record set, using row constructor
sSql := 'INSERT INTO myTable (myId,myCustomer,myValue) VALUES (¤1¤,$'¤2¤$',¤3¤),(¤4¤,$'¤5¤$',¤6¤)';

F_Replace(pString:= ADR(sSql), cbStringLen:= SIZEOF(sSql), sSearch:= '¤1¤', sReplace:= TO_STRING(aiId[0])); //Replace placeholder
F_Replace(pString:= ADR(sSql), cbStringLen:= SIZEOF(sSql), sSearch:= '¤2¤', sReplace:= asCustomer[0]); //Replace placeholder
F_Replace(pString:= ADR(sSql), cbStringLen:= SIZEOF(sSql), sSearch:= '¤3¤', sReplace:= TO_STRING(arValue[0])); //Replace placeholder

F_Replace(pString:= ADR(sSql), cbStringLen:= SIZEOF(sSql), sSearch:= '¤4¤', sReplace:= TO_STRING(aiId[1])); //Replace placeholder
F_Replace(pString:= ADR(sSql), cbStringLen:= SIZEOF(sSql), sSearch:= '¤5¤', sReplace:= asCustomer[1]); //Replace placeholder
F_Replace(pString:= ADR(sSql), cbStringLen:= SIZEOF(sSql), sSearch:= '¤6¤', sReplace:= TO_STRING(arValue[1])); //Replace placeholder



fbSql(
	bExecute:= bInsert, 
	wDBID:= 1, 
	pSql:= ADR(sSql), 
	cbSql:= SIZEOF(sSql), 
	pData:= 0, 
	cbData:= 0, 
	udiMaxOfRecord:= 0, 
	udiNoOfRecords=> , 
	bDone=> bDone, 
	bBusy=> , 
	bError=> bError, 
	sError=> sError);

END_PROGRAM

// ---- POUs/SQL/04_Update/P_SqlUpdate.TcPOU
PROGRAM P_SqlUpdate
VAR
	
	fbSql : FB_EasySql;
	sSql : STRING(1000);
		
	iId : INT; //Record to update
	sCustomer : STRING; //Data to update
	rValue : REAL; //Data to update
		
	bUpdate : BOOL; //Execute command
	bDone : BOOL; //Command done
	bError : BOOL; //Command error
	sError : STRING(255);
	
END_VAR

//Update record i database.
sSql := 'UPDATE alarmLog SET time = CURRENT_TIMESTAMP WHERE time = ¤1¤';

F_Replace(pString:= ADR(sSql), cbStringLen:= SIZEOF(sSql), sSearch:= '¤1¤', sReplace:= TO_STRING(P_SqlSelectAlarmLog.astData[0].dtTime));  //Replace placeholder
//F_Replace(pString:= ADR(sSql), cbStringLen:= SIZEOF(sSql), sSearch:= '¤2¤', sReplace:= TO_STRING(rValue)); //Replace placeholder
//F_Replace(pString:= ADR(sSql), cbStringLen:= SIZEOF(sSql), sSearch:= '¤3¤', sReplace:= TO_STRING(iId)); //Replace placeholder



fbSql(
	bExecute:= bUpdate, 
	wDBID:= 1, 
	pSql:= ADR(sSql), 
	cbSql:= SIZEOF(sSql), 
	pData:= 0, 
	cbData:= 0, 
	udiMaxOfRecord:= 0, 
	udiNoOfRecords=> , 
	bDone=> bDone, 
	bBusy=> , 
	bError=> bError, 
	sError=> sError);

END_PROGRAM

// ---- POUs/SQL/04_Update/P_SqlUpdateAlarmLog.TcPOU
PROGRAM P_SqlUpdateAlarmLog
VAR_INPUT
	bUpdate : BOOL; //Execute command
END_VAR
VAR
	
	fbSql : FB_EasySql;
	sSql : STRING(1000);
		
	iId : INT; //Record to update
	sCustomer : STRING; //Data to update
	rValue : REAL; //Data to update
		
	bDone : BOOL; //Command done
	bError : BOOL; //Command error
	sError : STRING(255);
	
END_VAR

//Update record i database.
sSql := 'UPDATE alarmLog SET alarmId = ¤1¤ WHERE time = (SELECT MAX( time ) FROM alarmLog );';

F_Replace(pString:= ADR(sSql), cbStringLen:= SIZEOF(sSql), sSearch:= '¤1¤', sReplace:= TO_STRING(P_SqlSelectAlarmLog.astData[0].alarmId));  //Replace placeholder
//F_Replace(pString:= ADR(sSql), cbStringLen:= SIZEOF(sSql), sSearch:= '¤2¤', sReplace:= TO_STRING(rValue)); //Replace placeholder
//F_Replace(pString:= ADR(sSql), cbStringLen:= SIZEOF(sSql), sSearch:= '¤3¤', sReplace:= TO_STRING(iId)); //Replace placeholder



fbSql(
	bExecute:= bUpdate, 
	wDBID:= 1, 
	pSql:= ADR(sSql), 
	cbSql:= SIZEOF(sSql), 
	pData:= 0, 
	cbData:= 0, 
	udiMaxOfRecord:= 0, 
	udiNoOfRecords=> , 
	bDone=> bDone, 
	bBusy=> , 
	bError=> bError, 
	sError=> sError);

END_PROGRAM

// ---- POUs/SQL/01_Insert/P_SqlInsertUnionAll.TcPOU
PROGRAM P_SqlInsertUnionAll
VAR
	
	fbSql : FB_EasySql;
	sSql : STRING(1000);
		
	aiId : ARRAY[0..1] OF INT; //Insert data
	asCustomer : ARRAY[0..1] OF STRING; //Insert data
	arValue : ARRAY[0..1] OF REAL; //Insert data
		
	bInsert : BOOL; //Execute command
	bDone : BOOL; //Command done
	bError : BOOL; //Command error
	sError : STRING(255);
	
END_VAR

// Insert more than one record, using UNION ALL, some databases execute UNION ALL faster than ROW CONSTRUCTOR
sSql := 'INSERT INTO myTable (myId,myCustomer,myValue) SELECT ¤1¤,$'¤2¤$',¤3¤ UNION ALL SELECT ¤4¤,$'¤5¤$',¤6¤';

F_Replace(pString:= ADR(sSql), cbStringLen:= SIZEOF(sSql), sSearch:= '¤1¤', sReplace:= TO_STRING(aiId[0])); //Replace placeholder
F_Replace(pString:= ADR(sSql), cbStringLen:= SIZEOF(sSql), sSearch:= '¤2¤', sReplace:= asCustomer[0]); //Replace placeholder
F_Replace(pString:= ADR(sSql), cbStringLen:= SIZEOF(sSql), sSearch:= '¤3¤', sReplace:= TO_STRING(arValue[0])); //Replace placeholder

F_Replace(pString:= ADR(sSql), cbStringLen:= SIZEOF(sSql), sSearch:= '¤4¤', sReplace:= TO_STRING(aiId[1])); //Replace placeholder
F_Replace(pString:= ADR(sSql), cbStringLen:= SIZEOF(sSql), sSearch:= '¤5¤', sReplace:= asCustomer[1]); //Replace placeholder
F_Replace(pString:= ADR(sSql), cbStringLen:= SIZEOF(sSql), sSearch:= '¤6¤', sReplace:= TO_STRING(arValue[1])); //Replace placeholder



fbSql(
	bExecute:= bInsert, 
	wDBID:= 1, 
	pSql:= ADR(sSql), 
	cbSql:= SIZEOF(sSql), 
	pData:= 0, 
	cbData:= 0, 
	udiMaxOfRecord:= 0, 
	udiNoOfRecords=> , 
	bDone=> bDone, 
	bBusy=> , 
	bError=> bError, 
	sError=> sError);

END_PROGRAM

// ---- POUs/SQL/02_Delete/P_SqlDelete.TcPOU
PROGRAM P_SqlDelete
VAR
	fbSql : FB_EasySql;
	sSql : STRING(1000);
		
	iId : INT; //ID to delete
	
	bDelete : BOOL; //Execute command
	bDone : BOOL; //Command done
	bError : BOOL; //Command error
	sError : STRING(255);
	
END_VAR

//Delete items from database
sSql := 'DELETE FROM myTable WHERE myId = ¤1¤';

F_Replace(pString:= ADR(sSql), cbStringLen:= SIZEOF(sSql), sSearch:= '¤1¤', sReplace:= TO_STRING(iId)); //Replace placeholder

fbSql(
	bExecute:= bDelete, 
	wDBID:= 1, 
	pSql:= ADR(sSql), 
	cbSql:= SIZEOF(sSql), 
	pData:= 0, 
	cbData:= 0, 
	udiMaxOfRecord:= 0, 
	udiNoOfRecords=> , 
	bDone=> bDone, 
	bBusy=> , 
	bError=> bError, 
	sError=> sError);

END_PROGRAM

// ---- POUs/SQL/05_Count/P_SqlCount.TcPOU
PROGRAM P_SqlCount
VAR
	
	fbSq : FB_EasySql;
	sSql : STRING(1000);
	
	sCustomer : STRING := 'Tom';
	
	diCount : LINT; //Data array for recieved data
	
	bCount : BOOL; //Execute command
	bDone : BOOL; //Command done
	bError : BOOL; //Command error
	sError : STRING(255);
	
	udiNoOfRecords : UDINT; //Numbers of returned recoreds
	
END_VAR

//Return record counts
sSql := 'SELECT COUNT(myCustomer) FROM myTable WHERE myCustomer = $'¤1¤$'';

F_Replace(pString:= ADR(sSql), cbStringLen:= SIZEOF(sSql), sSearch:= '¤1¤', sReplace:= sCustomer); //Replace placeholder

fbSq(
	bExecute:= bCount, 
	wDBID:= 1, 
	pSql:= ADR(sSql), 
	cbSql:= SIZEOF(sSql), 
	pData:= ADR(diCount), 
	cbData:= SIZEOF(diCount), 
	udiMaxOfRecord:= 1, //Max number of recieved records
	udiNoOfRecords=> udiNoOfRecords, 
	bDone=> bDone, 
	bBusy=> , 
	bError=> bError, 
	sError=> sError);

END_PROGRAM

// ---- POUs/SQL/06_Sum/P_SqlSum.TcPOU
PROGRAM P_SqlSum
VAR
	
	fbSq : FB_EasySql;
	sSql : STRING(1000);
	
	sCustomer : STRING := 'Tom';
	
	lrSum : LREAL; //Data for recieved data
	
	
	
	bSum : BOOL; //Execute command
	bDone : BOOL; //Command done
	bError : BOOL; //Command error
	sError : STRING(255);
	
	udiNoOfRecords : UDINT; //Numbers of returned recoreds
	
END_VAR

//Return sum of col.
sSql := 'SELECT SUM(myValue) FROM myTable WHERE myCustomer = $'¤1¤$'';

F_Replace(pString:= ADR(sSql), cbStringLen:= SIZEOF(sSql), sSearch:= '¤1¤', sReplace:= sCustomer); //Replace placeholder

fbSq(
	bExecute:= bSum, 
	wDBID:= 1, 
	pSql:= ADR(sSql), 
	cbSql:= SIZEOF(sSql), 
	pData:= ADR(lrSum), 
	cbData:= SIZEOF(lrSum), 
	udiMaxOfRecord:= 1, //Max number of recieved records
	udiNoOfRecords=> udiNoOfRecords, 
	bDone=> bDone, 
	bBusy=> , 
	bError=> bError, 
	sError=> sError);

END_PROGRAM

// ---- POUs/DB_Conn.TcPOU
PROGRAM DB_Conn
VAR
	iAlive: INT;
	frameSum : DINT;
	counter: INT;
END_VAR

iAlive := iAlive + 1;

IF P_SqlSelectRecipe.bDone THEN
	P_SqlSelectRecipe.bRead := FALSE;
	PROGRAM_DATA.uiCartheight		:= DINT_TO_UINT(P_SqlSelectRecipe.astData[0].recipe_cart_height);
	PROGRAM_DATA.uiValveDelay		:= DINT_TO_UINT(P_SqlSelectRecipe.astData[0].recipe_valve_delay);
	PROGRAM_DATA.usiImageRetryNo	:= DINT_TO_USINT(P_SqlSelectRecipe.astData[0].recipe_image_retry_no);
	PROGRAM_DATA.usiOpMode			:= DINT_TO_USINT(P_SqlSelectRecipe.astData[0].Operation_mode_id);
	PROGRAM_DATA.usiPackingPattern	:= DINT_TO_USINT(P_SqlSelectRecipe.astData[0].packing_pattern_id);
	PROGRAM_DATA.usiNewVelocity		:= DINT_TO_USINT(P_SqlSelectRecipe.astData[0].recipe_velocity);
END_IF

frameSum := FRAME_DATA.ct_x + FRAME_DATA.ct_y + FRAME_DATA.ct_z + FRAME_DATA.ct_a + FRAME_DATA.ct_e + FRAME_DATA.ct_r + 
			FRAME_DATA.pt_x + FRAME_DATA.pt_y + FRAME_DATA.pt_z + FRAME_DATA.pt_a + FRAME_DATA.pt_e + FRAME_DATA.pt_r + 
			FRAME_DATA.cw_x + FRAME_DATA.cw_y + FRAME_DATA.cw_z + FRAME_DATA.cw_a + FRAME_DATA.cw_e + FRAME_DATA.cw_r + 
			FRAME_DATA.pw_x + FRAME_DATA.pw_y + FRAME_DATA.pw_z + FRAME_DATA.pw_a + FRAME_DATA.pw_e + FRAME_DATA.pw_r;
IF P_SqlSelectFrame.bDone OR frameSum = 1 THEN
	P_SqlSelectFrame.bRead := TRUE;
	
	IF P_SqlSelectFrame.bDone THEN
		FOR counter:=0 TO 3 BY 1 DO
			IF P_SqlSelectFrame.astData[counter].sId = 'ct' THEN
				FRAME_DATA.ct_x := P_SqlSelectFrame.astData[counter].diX;
				FRAME_DATA.ct_y := P_SqlSelectFrame.astData[counter].diY;
				FRAME_DATA.ct_z := P_SqlSelectFrame.astData[counter].diZ;
				FRAME_DATA.ct_a := P_SqlSelectFrame.astData[counter].diA;
				FRAME_DATA.ct_e := P_SqlSelectFrame.astData[counter].diE;
				FRAME_DATA.ct_r := P_SqlSelectFrame.astData[counter].diR;
			ELSIF P_SqlSelectFrame.astData[counter].sId = 'pt' THEN
				FRAME_DATA.pt_x := P_SqlSelectFrame.astData[counter].diX;
				FRAME_DATA.pt_y := P_SqlSelectFrame.astData[counter].diY;
				FRAME_DATA.pt_z := P_SqlSelectFrame.astData[counter].diZ;
				FRAME_DATA.pt_a := P_SqlSelectFrame.astData[counter].diA;
				FRAME_DATA.pt_e := P_SqlSelectFrame.astData[counter].diE;
				FRAME_DATA.pt_r := P_SqlSelectFrame.astData[counter].diR;
			ELSIF P_SqlSelectFrame.astData[counter].sId = 'cw' THEN
				FRAME_DATA.cw_x := P_SqlSelectFrame.astData[counter].diX;
				FRAME_DATA.cw_y := P_SqlSelectFrame.astData[counter].diY;
				FRAME_DATA.cw_z := P_SqlSelectFrame.astData[counter].diZ;
				FRAME_DATA.cw_a := P_SqlSelectFrame.astData[counter].diA;
				FRAME_DATA.cw_e := P_SqlSelectFrame.astData[counter].diE;
				FRAME_DATA.cw_r := P_SqlSelectFrame.astData[counter].diR;
			ELSIF P_SqlSelectFrame.astData[counter].sId = 'pw' THEN
				FRAME_DATA.pw_x := P_SqlSelectFrame.astData[counter].diX;
				FRAME_DATA.pw_y := P_SqlSelectFrame.astData[counter].diY;
				FRAME_DATA.pw_z := P_SqlSelectFrame.astData[counter].diZ;
				FRAME_DATA.pw_a := P_SqlSelectFrame.astData[counter].diA;
				FRAME_DATA.pw_e := P_SqlSelectFrame.astData[counter].diE;
				FRAME_DATA.pw_r := P_SqlSelectFrame.astData[counter].diR;
			END_IF
		END_FOR;
		P_SqlSelectFrame.bRead := FALSE;
	END_IF
END_IF	

IF (PROGRAM_DATA.usiProgram = 0) OR (PROGRAM_DATA.usiRecipe = 0 ) THEN
	P_SqlSelectCurrent.bRead := TRUE;
	IF P_SqlSelectCurrent.bDone THEN
		P_SqlSelectCurrent.bRead 	:= FALSE;
		PROGRAM_DATA.usiNewProgram 	:= DINT_TO_USINT(P_SqlSelectCurrent.astData[0].program_no);
		PROGRAM_DATA.usiNewRecipe	:= DINT_TO_USINT(P_SqlSelectCurrent.astData[0].recipe_id);
		P_SqlSelectRecipe.bRead := TRUE;
	END_IF
END_IF

END_PROGRAM

// ---- POUs/OnOffRobotCut.TcPOU
PROGRAM OnOffRobotCut
VAR_INPUT
	State: INT := 0;
END_VAR


VAR



	uiSignalIn1 AT %I*: BYTE;		(* For running status PLC *)
	uiSignalIn3 AT %I*: BYTE;		(* For Online status *)

	(* Physical Botton on PLC box *)
	bStartBotton AT %I*: BOOL;

	NewState: INT := 0;
	StartUpRobot : BOOL;
	ShoutdownRobot : BOOL;

	(* Out *)
	bStart : BOOL;

	(*Timer*)
	TonWait : TON;

	byTest : ARRAY[0..1]OF BYTE;
	nTest : UINT;


	U1: BOOL;
END_VAR

(* Start connection to Robot Cut if physical botton or HMI button is pressed *)
IF bRobotConnect OR bStartBottonHMI THEN
	bRobotConnect := FALSE;
	StartUpRobot := TRUE;
END_IF

IF bRobotDisconnect THEN
	bRobotDisconnect := FALSE;
	ShoutdownRobot := TRUE;
END_IF

CASE State OF

	0:
		IF StartUpRobot AND NOT bStartNoHold THEN
			NewState  	:= 10;
		END_IF

		IF ShoutdownRobot AND NOT bNoDriveOff  THEN

			NewState  	:= 100;
		END_IF

		(*IF bAckAlarm THEN
			NewState := 200;
		END_IF*)

	10:(*NoHold And NoDriveOff*)
		bNoHold 	:= TRUE;
		bNoDriveOff	:= TRUE;

		IF TonWait.Q THEN
			NewState  := 20;
		END_IF

	20:(*Reset alarm*)
		GbCancelAlarm 	:= TRUE;

		IF bNoAlarm THEN
			NewState	:= 30;
		END_IF

	30:(*DriveOn*)
		GbCancelAlarm 	:= FALSE;
		bDriveOn 	:= TRUE;

		IF bDriveOnState THEN
			NewState  	:= 40;
		END_IF

	40:(*Start*)
		GbCancelAlarm := FALSE;
		bStart := TRUE;

		IF bStartNoHold THEN
			NewState  	:= 50;
		END_IF

	50:(*DONE StartUp*)
		bStart 		:= FALSE;
		StartUpRobot := FALSE;
		NewState  	:= 0;

	100:
		bNoHold		:= FALSE;

		IF NOT bStartNoHold THEN
			NewState  	:=110 ;
		END_IF

	110:
		bNoHold		:= TRUE;
		bNoDriveOff	:= FALSE;

		IF NOT bDriveOnState THEN
			NewState  	:=120 ;
		END_IF

	120: (*DONE Shoutdown *)
		bNoDriveOff		:= TRUE;
		ShoutdownRobot 	:= FALSE;
		NewState  	:=0 ;

	200:

		IF NOT bDriveOnState THEN
			bDriveOn := FALSE;
			IF TonWait.Q THEN
				NewState  := 210;
			END_IF
		ELSE
			NewState := 0;
		END_IF

	210:
		(* Reset, og gør klar til at køre igen *)
		bDriveOn := TRUE;
		IF TonWait.Q THEN
			uiStatus := 0;
			NewState  := 0;
		END_IF



END_CASE

uiSignalOut1.00 := bDriveOn;
uiSignalOut1.01 := bNoDriveOff;
uiSignalOut1.02 := bStart;
uiSignalOut1.03 := bNoHold;
uiSignalOut1.04 := U1;
uiSignalOut2.00 := GbCancelAlarm;


(* Check if devices are running *)

NewbPLCStatus := TRUE;
IF uiSignalIn3.01 THEN
	NewbRobotCutStatus := TRUE;
ELSE
	NewbRobotCutStatus := FALSE;
END_IF
IF uiSignalIn3.00 = TRUE THEN
	NewbRobotPickStatus := TRUE;
ELSE
	NewbRobotPickStatus := FALSE;
END_IF


bNoAlarm 		:= uiSignalIn1.00;
bDriveOnState	:= uiSignalIn1.01;
bStartNoHold		:= uiSignalIn1.02;

TonWait(IN:=State = 10 OR State = 200,	PT:=t#1000ms ,	Q=> ,	ET=> );

END_PROGRAM

// ---- POUs/LogProgram.TcPOU
PROGRAM LogProgram
VAR_INPUT
	State: INT :=0;
	NewState: INT := 0;

END_VAR

VAR
	bStart: BOOL;		// Start the sequence
END_VAR

///////////////////////////// For logging of datas /////////////////////////////
IF bLog THEN
	bStart := TRUE;
	
ELSE 
	bStart := FALSE;
END_IF

CASE State OF

	0:	
		tLogTime.IN 		:= FALSE;
		uiElapsedTime		:= 0;
		usiImageLog			:= 0;
		usiStickoutCutLog	:= 0;
		usiRetryLog			:= 0;
		usiImageRetry		:= 0;
		bLogSucces			:= 0;
		IF bStart THEN
			bStart := FALSE;
			tLogTime.IN := TRUE;
			NewState := 10;
		END_IF
		
	10:		// Check if all states are in state 0	-	This means that the sequence has finished
		IF (Tools.State = 0) AND (Control.State = 0) THEN
			bLog := FALSE;
			uiElapsedTime := TO_UINT(tLogTime.ET);
			NewState := 20;
		END_IF 
		
	20:
		P_SqlInsertLog.bInsert := TRUE;
		IF P_SqlInsertLog.bDone THEN
			P_SqlInsertLog.bInsert := FALSE;
			NewState := 0;
		END_IF

END_CASE


(*
	bLog:				BOOL;		// For logging of data
	tLogTime:			TON;		// Time for one sequence
	usiImageLog:		USINT;		// Counting number of images taken in a sequence
	usiStickoutCutLog:	USINT;		// For counting number of stick-outs
	bLogSucces:			BOOL;		// TRUE if success	-	FALSE if not
*)

///////////////////////////// Timers /////////////////////////////
tLogTime (PT := T#5M);

END_PROGRAM

// ---- POUs/Tools.TcPOU
PROGRAM Tools
VAR_INPUT
	State: INT :=0;
	NewState: INT := 0;

END_VAR

VAR


	bValveTime: BOOL;
	bDriveTime: BOOL;
	bDriveTime2: BOOL;
	bSaveData: BOOL := 0;

	(* uiStepsToMove			-->	Antal pulser på tællerkort	:	24 Pulser pr mm * antal mm	*)
	uiStepsToMove: UINT := 0;

	(*Inputs*)


	(*Outputs*)
	bValve1Control : BOOL;
	qValve1 AT %Q*: BOOL := FALSE;		(* Ventil 1 --> Load Cutter 			*)
	qValve2	AT %Q*:BOOL := FALSE;		(* Ventil 2 --> Kører stempel i cut op		*)
	qValve3	AT %Q*:BOOL := FALSE;		(* Ventil 3 --> Brake 				*)
	qValve4	AT %Q*:BOOL := FALSE;		(* Ventil 4 --> Luk Gripper			*)
	qValve5 AT %Q*:BOOL := FALSE;		(* Ventil 5 --> Picker  				*)

	qMotorRun AT %Q*:BOOL := FALSE;		(* Gripper arm ind					*)
	qMotorDirection AT %Q*: BOOL := FALSE;		(* Gripper arm ud					*)

	(*Triggers*)
	bBtnPress: R_TRIG;

	(*Timer*)
	WaitValve:TON;
	WaitMotorDrive: TON;
	WaitMotorDrive2: TON;
	encoderSteps: INT := 5;
	InOrOut: BOOL;
	maxValue: UDINT;
	minValue: UDINT;
	temp: BOOL;
	timer: TON;
	timer2: INT := 0;
	testing: BOOL;
	stepValue: UDINT;
	next: BOOL;
	WaitGrip2: TON;
	bWaitGrip2: BOOL;
	bWaitGrip: BOOL;
	testStart: BOOL;
	bReset: BOOL;
	OnTime: UINT := 150;
	OffTime: UINT := 150;
	tonBlinkOn: TON;
	tonBlinkOff: TON;
	flag: BOOL;
	Wait: TON;
	bWait: BOOL;
	bPickOpened: BOOL;
	bCutOpened: BOOL;
	bCutDeloaded: BOOL;
	bBladesDown: BOOL;
	bLoadReleased: BOOL;
	bGripOpened: BOOL;
	bGripHome: BOOL;
	bOut: BOOL := TRUE;
	bIn: BOOL := FALSE;
	Wait2: TON;
	bWait2: BOOL;
	bStopped: BOOL;
	bValve4Control: BOOL;
	bbFlag: BOOL;
	resetCount: UINT := 0;
	
	tempTime : STRING(255);
	brakeOn: BOOL;
	TEST: BOOL;
END_VAR

CASE State OF

	0:	(* Check hvilken kommando udføre *)
		bValveTime := FALSE;
		bSaveData := FALSE;
		bAck := FALSE;						(* Acknowledge to control programs, that the tool operation has been executed *)

		(* --------- RobotGrip --------- *)

		IF GbGripStem THEN
			GbGripStem	:= FALSE;
			bAck := TRUE;
			NewState	:= 100;
		END_IF

		IF GbReleaseStem THEN
			GbReleaseStem	:= FALSE;
			bAck := TRUE;
			NewState	:= 150;
		END_IF

		IF GbHomeGripStem OR (sToolControl = 'grip-home') THEN
			GbHomeGripStem	:= FALSE;
			bAck := TRUE;
			NewState	:= 200;
		END_IF

	(* -------------------------------------------------------------------------------- 		Grip		 -------------------------------------------------------------------------------- *)
	(* ---------------------------------------- 	Grab stem and Pull in 	 ---------------------------------------- *)

	100:		(*  MotorOut untill the encoder count Reaches *)

		(* Direction TRUE	-->	Move in *)
		(* Direction FALSE	-->	Move out *)
		qMotorDirection := bOut;
		qMotorRun := TRUE;
		(* uiSignalInEncoderCount	-->	Antal pulser på tællerkort	: 	10 000 pulser = grip helt inde						*)
		(* uiStepsToMove			-->	Antal pulser på tællerkort	:	24 Pulser pr mm * antal mm 						*)
		(* uiSetCounterValue		-->	Max antal pulser			:	Når  uiSignalInEncoderCount = 0, er grip helt ude.	*)
		IF uiSignalInEncoderCount < (uiSetCounterValue - uiStepsToMove) THEN
			qMotorRun := FALSE;
			(* minValue		-->	Der hvor gripper endte *)
			minValue := uiSignalInEncoderCount;
			NewState 	:= 110;
		END_IF

	110:		(*  Close grip *)
		qValve4 := TRUE;
		bValveTime := TRUE;

		IF waitValve.Q THEN
			bValveTime := FALSE;
			NewState 	:=120;
		END_IF

		
	120:
		(* stepValue		-->	Offset der blev skabt da der kørtes ud *)
		IF NOT qMotorRun THEN
			stepValue := uiSetCounterValue - (minValue - uiSignalInEncoderCount);		(* Slack distance the arm moves too far - Used for when moving back In *) (* + 60 *)
		END_IF

		qMotorDirection := bIn;
		qMotorRun := TRUE;

		(* bGripSensorStop	-->	Endestop					: 	Bruges til Homing						*)
		(* maxValue			-->	Offset fra at bevæge arm ind	: 	Bruges til når planten igen skal afleveres	*)
		IF  bGripSensorStop OR uiSignalInEncoderCount >= stepValue THEN
			qMotorRun := FALSE;
			maxValue := uiSignalInEncoderCount;

			bWait2 := TRUE;
			IF Wait2.Q THEN
				bWait2 := FALSE;
				NewState 	:=0;
			END_IF
		END_IF

	(* ---------------------------------------- 	Release stem	 ---------------------------------------- *)
	150:

		(* Direction TRUE	-->	Move in *)
		(* Direction FALSE	-->	Move out *)
		qMotorDirection := bOut;
		qMotorRun := TRUE;


		(* uiSignalInEncoderCount	-->	Antal pulser på tællerkort	: 	10 000 pulser = grip helt inde						*)
		(* uiStepsToMove			-->	Antal pulser på tællerkort	:	24 Pulser pr mm * antal mm 						*)
		(* uiSetCounterValue		-->	Max antal pulser			:	Når  uiSignalInEncoderCount = 0, er grip helt ude.	*)
		IF uiSignalInEncoderCount < (uiSetCounterValue - uiStepsToMove) THEN
			qMotorRun := FALSE;
			(* minValue		-->	Der hvor gripper endte *)
			minValue := uiSignalInEncoderCount;
			NewState 	:= 160;
		END_IF

	160:		(* Release the Stem *)

		qValve4 := FALSE;
		bValveTime := TRUE;

		IF waitValve.Q THEN
			bValveTime := FALSE;
			NewState 	:=170;
		END_IF

	170:
		(* stepValue		-->	Offset der blev skabt da der kørtes ud *)
		IF NOT qMotorRun THEN
			stepValue := uiSetCounterValue - (minValue - uiSignalInEncoderCount);		(* Slack distance the arm moves too far - Used for when moving back In *)
		END_IF

		qMotorDirection := bIn;
		qMotorRun := TRUE;

		(* bGripSensorStop	-->	Endestop					: 	Bruges til Homing						*)
		(* maxValue			-->	Offset fra at bevæge arm ind	: 	Bruges til når planten igen skal afleveres	*)
		IF  bGripSensorStop OR uiSignalInEncoderCount >= stepValue THEN
			qMotorRun := FALSE;
			maxValue := uiSignalInEncoderCount;
			bWait2 := TRUE;
			IF Wait2.Q THEN
				bWait2 := FALSE;
				NewState 	:=0;
			END_IF
		END_IF

	(* ---------------------------------------- 	Homing Grip 	 ---------------------------------------- *)
	200:		(* Homing *)
		IF  bGripSensorStop THEN
			bSetCounter := FALSE;
			qMotorRun := FALSE;
			bDriveTime := TRUE;
			IF WaitMotorDrive.Q THEN
				bSetCounter := TRUE;
				bDriveTime := FALSE;
				bHomeDone := TRUE;
				NewState 	:= 0;
			END_IF
		ELSE
			qMotorDirection := bIn;
			qMotorRun := TRUE;
		END_IF

	1000:	(* RESET *)
		IF NOT bbFlag THEN
			bAck := FALSE;
			bbFlag := TRUE;
			resetCount := 0;
		END_IF

		(* Først Åben Pick *)
		IF resetCount = 0 THEN
			FB_OPEN_PICK.Execute := TRUE;
			resetCount := resetCount + 1;
		END_IF
		IF FB_OPEN_PICK.Done THEN
			bPickOpened := TRUE;
			FB_OPEN_PICK.Execute := FALSE;
		END_IF

		(* Åben Cut *)
		IF resetCount = 1 THEN
			FB_OPEN_CUT.Execute := TRUE;
			resetCount := resetCount + 1;
		END_IF
		IF FB_OPEN_CUT.Done THEN
			bCutOpened := TRUE;
			FB_OPEN_CUT.Execute := FALSE;
		END_IF

		(* Deload Cut *)
		IF resetCount = 2 THEN
			FB_DELOAD_CUT.Execute := TRUE;
			resetCount := resetCount + 1;
		END_IF
		IF FB_DELOAD_CUT.Done THEN
			bCutDeloaded := TRUE;
			FB_DELOAD_CUT.Execute := FALSE;
			resetCount := 0;
		END_IF

		(* Open Grip *)
		IF bCutOpened AND NOT bGripOpened THEN
			qValve4 := FALSE;
			bGripOpened := TRUE;
		END_IF

		IF bGripOpened AND NOT bGripHome THEN
			IF  bGripSensorStop THEN
				bSetCounter := FALSE;
				qMotorRun := FALSE;
				bDriveTime := TRUE;
				IF WaitMotorDrive.Q THEN
					bSetCounter := TRUE;
					bDriveTime := FALSE;
					bGripHome := TRUE;
				END_IF
			ELSE
				qMotorDirection := bIn;
				qMotorRun := TRUE;
			END_IF
		END_IF

		IF bPickOpened AND bCutOpened AND bCutDeloaded AND bGripOpened AND bGripHome AND NOT bAck THEN
			FB_OPEN_CUT.		Execute := FALSE;
			FB_CLOSE_CUT.		Execute := FALSE;
			FB_RELEASE_CUT.		Execute := FALSE;
			FB_OPEN_PICK.		Execute := FALSE;
			FB_CLOSE_PICK.		Execute := FALSE;
			FB_LOAD_CUT.		Execute := FALSE;
			FB_DELOAD_CUT.		Execute := FALSE;
			FB_OPEN_GRIP.		Execute := FALSE;
			FB_CLOSE_GRIP.		Execute := FALSE;


			GbDeloadCut 	:= FALSE;
			GbOpenCut 		:= FALSE;
			GbOpenPick 		:= FALSE;

			bLoadReleased 	:= FALSE;
			bBladesDown 	:= FALSE;

			bPickOpened 	:= FALSE;
			bCutOpened 		:= FALSE;
			bCutDeloaded 	:= FALSE;
			bGripOpened 	:= FALSE;
			bGripHome 		:= FALSE;
			bAck 			:= FALSE;
			bbFlag 			:= FALSE;
			NewState 		:= 0;
		END_IF

	2000:
		bStopped := TRUE;


	3000:	(* RESET *)
		IF NOT bbFlag THEN
			bAck := FALSE;
			bbFlag := TRUE;
		END_IF

		(* Først Åben Pick *)
		GbOpenPick := TRUE;
		IF FB_OPEN_PICK.Done THEN
			bPickOpened := TRUE;
			GbOpenPick := FALSE;
		END_IF

		(* Åben Cut *)
		GbOpenCut := TRUE;
		IF FB_OPEN_CUT.Done THEN
			bCutOpened := TRUE;
			GbOpenCut := FALSE;
		END_IF

		(* Open Grip *)
		IF bCutOpened AND NOT bGripOpened THEN
			qValve4 := FALSE;
			bGripOpened := TRUE;
		END_IF

		IF bGripOpened AND NOT bGripHome THEN
			IF  bGripSensorStop THEN
				bSetCounter := FALSE;
				qMotorRun := FALSE;
				bDriveTime := TRUE;
				IF WaitMotorDrive.Q THEN
					bSetCounter := TRUE;
					bDriveTime := FALSE;
					bGripHome := TRUE;
				END_IF
			ELSE
				qMotorDirection := bIn;
				qMotorRun := TRUE;
			END_IF
		END_IF

		IF bPickOpened AND bCutOpened AND bGripOpened AND bGripHome AND NOT bAck THEN
			FB_OPEN_CUT.		Execute := FALSE;
			FB_CLOSE_CUT.		Execute := FALSE;
			FB_RELEASE_CUT.	Execute := FALSE;
			FB_OPEN_PICK.		Execute := FALSE;
			FB_CLOSE_PICK.		Execute := FALSE;
			FB_LOAD_CUT.		Execute := FALSE;
			FB_DELOAD_CUT.	Execute := FALSE;
			FB_OPEN_GRIP.		Execute := FALSE;
			FB_CLOSE_GRIP.		Execute := FALSE;


			GbDeloadCut := FALSE;
			GbOpenCut := FALSE;
			GbOpenPick := FALSE;

			bLoadReleased := FALSE;
			bBladesDown := FALSE;

			bPickOpened := FALSE;
			bCutOpened := FALSE;
			bCutDeloaded := FALSE;
			bGripOpened := FALSE;
			bGripHome := FALSE;
			bAck := FALSE;
			bbFlag := FALSE;
			NewState := 0;
		END_IF

END_CASE

IF bReset THEN
	bReset := FALSE;
	NewState := 0;
END_IF

IF State <> 2000 THEN
	bStopped := FALSE;
END_IF

tempTime := CONCAT ('T#', UINT_TO_STRING(PROGRAM_DATA.uiValveDelay));

